METHOD PUBLIC CallAfterInit
VAR_INPUT
    AxisRef : REFERENCE TO AXIS_REF;
END_VAR
THIS^.AxisRef REF= AxisRef;
END_METHOD

{warning 'add property implementation'}
PROPERTY Done : BOOL
GET
Done := bDone;
END_GET
END_PROPERTY

{warning 'add property implementation'}
PROPERTY Error : BOOL
GET
Error := bError;
END_GET
END_PROPERTY

{warning 'add property implementation'}
PROPERTY ErrorID : UDINT
GET
ErrorID := nErrorID;
END_GET
END_PROPERTY

METHOD FB_Init : BOOL
VAR_INPUT
    bInitRetains : BOOL; // if TRUE, the retain variables are initialized (warm start / cold start)
    bInCopyCode : BOOL;  // if TRUE, the instance afterwards gets moved into the copy code (online change)
    AxisRef : REFERENCE TO AXIS_REF;
END_VAR
THIS^.AxisRef REF= AxisRef;
END_METHOD

PROPERTY Message : T_MAXSTRING
GET
Message :=sMessage;
END_GET
END_PROPERTY

METHOD Reset
VAR_INPUT
    Execute	: BOOL;
END_VAR
THIS^.bExecute := Execute;
END_METHOD

END_FUNCTION_BLOCK

// ---- POUs/FBs/NC/FB_HaltNC.TcPOU
FUNCTION_BLOCK FB_HaltNC IMPLEMENTS I_Halt
VAR_INPUT
    {attribute 'no_copy'}
    AxisRef : REFERENCE TO AXIS_REF;
    fbMcHalt 		: MC_Halt;
    bCommandHalt :BOOL;
    fDeceleration : LREAL;
    fJerk :LREAL;
    eBufferMode : MC_BufferMode := MC_BufferMode.MC_Aborting;
    bError : BOOL;
    bBusy : BOOL;
    bDone : BOOL;
    nErrorID : UDINT;
    sMessage : T_MAXSTRING;
    rtDone : R_TRIG;
    bAborted : BOOL;
END_VAR
VAR_OUTPUT
END_VAR
VAR
END_VAR

IF NOT __ISVALIDREF(THIS^.AxisRef) THEN
    RETURN;
END_IF

THIS^.AxisRef.ReadStatus();

THIS^.fbMcHalt(
    Axis := THIS^.AxisRef,
    Execute := THIS^.bCommandHalt,
    Deceleration := THIS^.fDeceleration,
    Jerk := THIS^.fJerk,
    BufferMode := THIS^.eBufferMode,
    Done =>THIS^.bDone,
    Busy => THIS^.bBusy,
    CommandAborted =>THIS^.bAborted,
    Error => THIS^.bError,
    ErrorID => THIS^.nErrorID
);

rtDone(CLK:=bDone);
IF  rtDone.Q THEN
    THIS^.bCommandHalt := FALSE;
END_IF

{warning 'Add property implementation'}
PROPERTY Aborted : BOOL
GET
Aborted := THIS^.bAborted;
END_GET
END_PROPERTY

{warning 'Add property implementation'}
PROPERTY Active : BOOL
GET
Active := THIS^.fbMcHalt.Active;
END_GET
END_PROPERTY

{warning 'add property implementation'}
PROPERTY Busy : BOOL
GET
Busy := bBusy;
END_GET
END_PROPERTY

METHOD PUBLIC CallAfterInit
VAR_INPUT
    AxisRef : REFERENCE TO AXIS_REF;
END_VAR
THIS^.AxisRef REF= AxisRef;
END_METHOD

PROPERTY CommandHalt : BOOL
SET
bCommandHalt := CommandHalt;
END_SET
END_PROPERTY

PROPERTY Done : BOOL
GET
Done := bDone;
END_GET
END_PROPERTY

{warning 'add property implementation'}
PROPERTY Error : BOOL
GET
Error := bError;
END_GET
END_PROPERTY

{warning 'add property implementation'}
PROPERTY ErrorID : UDINT
GET
ErrorID := nErrorID;
END_GET
END_PROPERTY

//FB_Init is always available implicitly and it is used primarily for initialization.
//The return value is not evaluated. For a specific influence, you can also declare the
//methods explicitly and provide additional code there with the standard initialization
//code. You can evaluate the return value.
METHOD FB_Init: BOOL
VAR_INPUT
    bInitRetains: BOOL; // TRUE: the retain variables are initialized (reset warm / reset cold)
    bInCopyCode: BOOL;  // TRUE: the instance will be copied to the copy code afterward (online change)
    AxisRef : REFERENCE TO AXIS_REF;
END_VAR
THIS^.AxisRef REF= AxisRef;
END_METHOD

METHOD Halt
VAR_INPUT
    Execute	: BOOL;
    Deceleration	: LREAL := 0;
    Jerk	: LREAL := 0;
    BufferMode	: MC_BufferMode := .MC_BufferMode.MC_Aborting;
END_VAR
THIS^.bCommandHalt :=  Execute;
THIS^.fDeceleration := Deceleration;
THIS^.fJerk := Jerk;
THIS^.eBufferMode := BufferMode;
END_METHOD

PROPERTY Message : T_MAXSTRING
GET
Message  := sMessage;
END_GET
END_PROPERTY

END_FUNCTION_BLOCK

// ---- Test/NC/FB_MotionAxisNC_Test.TcPOU
FUNCTION_BLOCK FB_MotionAxisNC_Test EXTENDS FB_TestSuite
VAR
	fbAxisRef : AXIS_REF;
	fbMotionLogger : FB_MotionLogger;
    fbHome : FB_HomeNC_TestDouble;
    fbHalt : FB_HaltNC_TestDouble;
    fbPower : FB_PowerNC_TestDouble;
    fbReset : FB_ResetNC_TestDouble;
    fbMoveAbsolute : FB_MoveAbsoluteNC_TestDouble;
    fbReadParameter : FB_ReadParameterNC_TestDouble;
    fbWriteParameter  : FB_WriteParameterNC_TestDouble;
    fbParamSaveRestore: FB_ParamSaveRestoreNC_TestDouble;
    fbEncoderScaling : FB_EncoderScalingNC_TestDouble;
    fbAxisStatus : FB_AxisStatusNC_TestDouble;
    fbBacklashCompensation : FB_BacklashCompensationNC_TestDouble;
END_VAR

GivenAllMCBlockErrorConditionThenPowerErrorHasHigherPriority();

METHOD PRIVATE GivenAllMCBlockErrorConditionThenPowerErrorHasHigherPriority
VAR_INST
    // subject under test
    // subject under test
    fbMotionAxis : FB_MotionAxisNC(  	
		AxisRef :=fbAxisRef,
		iMotionLogger := fbMotionLogger,
		iHome := fbHome,
        iHalt := fbHalt,
        iPower := fbPower,
        iReset := fbReset,
        iMoveAbsolute := fbMoveAbsolute,
        iReadParameter := fbReadParameter,
        iWriteParameter  := fbWriteParameter,
        iParamsSaveRestore:= fbParamSaveRestore,
        iEncoderScaling := fbEncoderScaling,
        iBacklashCompensation := fbBacklashCompensation
	);
bExpectedAxisError :BOOL := TRUE;
nExpectedErrorId: UDINT;
END_VAR
TEST(__POUNAME());
// ----- Power: Highest priority -----
fbHome.Error := TRUE;
fbHalt.Error := TRUE;
fbPower.Error := TRUE;
fbReset.Error := TRUE;
fbMoveAbsolute.Error := TRUE;
fbReadParameter.Error := TRUE;
fbWriteParameter.Error := TRUE;
fbParamSaveRestore.Error := TRUE;
fbBacklashCompensation.Error := TRUE;

fbMotionAxis();

AssertTrue(
    Condition := fbMotionAxis.Status.bError,
    Message   := 'Prioritized and generalized Error must be set #1'
);
AssertEquals_UDINT(
    Expected := 18000,
    Actual   := fbMotionAxis.Status.nErrorID,
    Message  := 'Prioritized error Id must be 18000 #2'
);

// ----- Halt: Second -----
fbPower.Error := FALSE;
fbHalt.Error := TRUE;
fbHome.Error := TRUE;
fbReset.Error := TRUE;
fbMoveAbsolute.Error := TRUE;
fbReadParameter.Error := TRUE;
fbWriteParameter.Error := TRUE;
fbParamSaveRestore.Error := TRUE;
fbBacklashCompensation.Error := TRUE;

fbMotionAxis();

AssertTrue(
    Condition := fbMotionAxis.Status.bError,
    Message   := 'Prioritized and generalized Error must be set #3'
);
AssertEquals_UDINT(
    Expected := 19000,
    Actual   := fbMotionAxis.Status.nErrorID,
    Message  := 'Prioritized error Id must be 19000 #4'
);

// ----- Reset: Third -----
fbPower.Error := FALSE;
fbHalt.Error := FALSE;
fbReset.Error := TRUE;
fbHome.Error := TRUE;
fbMoveAbsolute.Error := TRUE;
fbReadParameter.Error := TRUE;
fbWriteParameter.Error := TRUE;
fbParamSaveRestore.Error := TRUE;
fbBacklashCompensation.Error := TRUE;

fbMotionAxis();

AssertTrue(
    Condition := fbMotionAxis.Status.bError,
    Message   := 'Prioritized and generalized Error must be set #5'
);
AssertEquals_UDINT(
    Expected := 20000,
    Actual   := fbMotionAxis.Status.nErrorID,
    Message  := 'Prioritized error Id must be 20000 #6'
);

// ----- BacklashCompensation: Fourth -----
fbPower.Error := FALSE;
fbHalt.Error := FALSE;
fbReset.Error := FALSE;
fbBacklashCompensation.Error := TRUE;
fbHome.Error := TRUE;
fbMoveAbsolute.Error := TRUE;
fbReadParameter.Error := TRUE;
fbWriteParameter.Error := TRUE;
fbParamSaveRestore.Error := TRUE;

fbMotionAxis();

AssertTrue(
    Condition := fbMotionAxis.Status.bError,
    Message   := 'Prioritized and generalized Error must be set #7'
);
AssertEquals_UDINT(
    Expected := 21000,
    Actual   := fbMotionAxis.Status.nErrorID,
    Message  := 'Prioritized error Id must be 21000 #8'
);

// ----- MoveAbsolute: Fifth -----
fbBacklashCompensation.Error := FALSE;
fbMoveAbsolute.Error := TRUE;
fbPower.Error := FALSE;
fbHalt.Error := FALSE;
fbReset.Error := FALSE;
fbHome.Error := TRUE;
fbReadParameter.Error := TRUE;
fbWriteParameter.Error := TRUE;
fbParamSaveRestore.Error := TRUE;

fbMotionAxis();

AssertTrue(
    Condition := fbMotionAxis.Status.bError,
    Message   := 'Prioritized and generalized Error must be set #9'
);
AssertEquals_UDINT(
    Expected := 22000,
    Actual   := fbMotionAxis.Status.nErrorID,
    Message  := 'Prioritized error Id must be 22000 #10'
);

// ----- Home: Sixth -----
fbMoveAbsolute.Error := FALSE;
fbHome.Error := TRUE;
fbPower.Error := FALSE;
fbHalt.Error := FALSE;
fbReset.Error := FALSE;
fbBacklashCompensation.Error := FALSE;
fbReadParameter.Error := TRUE;
fbWriteParameter.Error := TRUE;
fbParamSaveRestore.Error := TRUE;

fbMotionAxis();

AssertTrue(
    Condition := fbMotionAxis.Status.bError,
    Message   := 'Prioritized and generalized Error must be set #11'
);
AssertEquals_UDINT(
    Expected := 23000,
    Actual   := fbMotionAxis.Status.nErrorID,
    Message  := 'Prioritized error Id must be 23000 #12'
);

// ----- ReadParameter: Eighth -----
fbHome.Error := FALSE;
fbReadParameter.Error := TRUE;
fbWriteParameter.Error := TRUE;
fbPower.Error := FALSE;
fbHalt.Error := FALSE;
fbReset.Error := FALSE;
fbBacklashCompensation.Error := FALSE;
fbMoveAbsolute.Error := FALSE;
fbParamSaveRestore.Error := TRUE;

fbMotionAxis();

AssertTrue(
    Condition := fbMotionAxis.Status.bError,
    Message   := 'Prioritized and generalized Error must be set #13'
);
AssertEquals_UDINT(
    Expected := 25000,
    Actual   := fbMotionAxis.Status.nErrorID,
    Message  := 'Prioritized error Id must be 25000 #14'
);

// ----- WriteParameter: Ninth -----
fbReadParameter.Error := FALSE;
fbWriteParameter.Error := TRUE;
fbPower.Error := FALSE;
fbHalt.Error := FALSE;
fbReset.Error := FALSE;
fbBacklashCompensation.Error := FALSE;
fbMoveAbsolute.Error := FALSE;
fbHome.Error := FALSE;
fbParamSaveRestore.Error := TRUE;

fbMotionAxis();

AssertTrue(
    Condition := fbMotionAxis.Status.bError,
    Message   := 'Prioritized and generalized Error must be set #15'
);
AssertEquals_UDINT(
    Expected := 26000,
    Actual   := fbMotionAxis.Status.nErrorID,
    Message  := 'Prioritized error Id must be 26000 #16'
);

// ----- ParamSaveRestore: Tenth -----
fbWriteParameter.Error := FALSE;
fbParamSaveRestore.Error := TRUE;
fbPower.Error := FALSE;
fbHalt.Error := FALSE;
fbReset.Error := FALSE;
fbBacklashCompensation.Error := FALSE;
fbMoveAbsolute.Error := FALSE;
fbHome.Error := FALSE;
fbReadParameter.Error := FALSE;

fbMotionAxis();

AssertTrue(
    Condition := fbMotionAxis.Status.bError,
    Message   := 'Prioritized and generalized Error must be set #17'
);
AssertEquals_UDINT(
    Expected := 27000,
    Actual   := fbMotionAxis.Status.nErrorID,
    Message  := 'Prioritized error Id must be 27000 #18'
);

TEST_FINISHED();
END_METHOD

END_FUNCTION_BLOCK

// ---- Test/TestDouble/FB_HomeNC_TestDouble.TcPOU
FUNCTION_BLOCK FB_HomeNC_TestDouble IMPLEMENTS I_Home
VAR
    bError : BOOL;
    nErrorID : UDINT := 23000;
END_VAR

PROPERTY Aborted : BOOL
GET
END_GET
END_PROPERTY

{warning 'Add method implementation '}
METHOD AbortRecovery
END_METHOD

PROPERTY Active : BOOL
GET
END_GET
END_PROPERTY

PROPERTY Busy : BOOL
GET
END_GET
END_PROPERTY

{warning 'Add method implementation '}
METHOD ClearStatus
END_METHOD

PROPERTY Done : BOOL
GET
END_GET
END_PROPERTY

PROPERTY Error : BOOL
GET
Error := bError;
END_GET
SET
bError := Error;
END_SET
END_PROPERTY

PROPERTY ErrorID : UDINT
GET
ErrorId := nErrorID;
END_GET
SET
nErrorId := ErrorID;
END_SET
END_PROPERTY

METHOD Home : BOOL
VAR_INPUT
    Position        : LREAL         := DEFAULT_HOME_POSITION;
    BufferMode      : MC_BufferMode;
 	HomeMode: INT :=E_EpicsHomeCmd.NONE;
END_VAR
END_METHOD

{warning 'Add method implementation '}
METHOD HomeDone
END_METHOD

PROPERTY LimHomeDone : BOOL
GET
END_GET
END_PROPERTY

PROPERTY Message : T_MAXSTRING
GET
END_GET
END_PROPERTY

PROPERTY Mode : INT
GET
END_GET
SET
END_SET
END_PROPERTY

PROPERTY Offset : LREAL
SET
END_SET
END_PROPERTY

PROPERTY Position : LREAL
SET
END_SET
END_PROPERTY

END_FUNCTION_BLOCK

// ---- Test/TestDouble/FB_HaltNC_TestDouble.TcPOU
FUNCTION_BLOCK FB_HaltNC_TestDouble IMPLEMENTS  I_Halt
VAR
	bError : BOOL;
	nErrorID : UDINT := 19000;
END_VAR

{warning 'Add property implementation'}
PROPERTY Aborted : BOOL
GET
END_GET
END_PROPERTY

{warning 'Add property implementation'}
PROPERTY Active : BOOL
GET
Active := TRUE;
END_GET
END_PROPERTY

{warning 'Add property implementation'}
PROPERTY Busy : BOOL
GET
END_GET
END_PROPERTY

{warning 'Add property implementation'}
PROPERTY CommandHalt : BOOL
SET
END_SET
END_PROPERTY

{warning 'Add property implementation'}
PROPERTY Done : BOOL
GET
END_GET
END_PROPERTY

{warning 'Add property implementation'}
PROPERTY Error : BOOL
GET
Error := bError;
END_GET
SET
bError := Error;
END_SET
END_PROPERTY

{warning 'Add property implementation'}
PROPERTY ErrorID : UDINT
GET
ErrorId := nErrorID;
END_GET
SET
nErrorId := ErrorID;
END_SET
END_PROPERTY

{warning 'Add method implementation '}
METHOD Halt
VAR_INPUT
	Deceleration	: LREAL := 0;
	Jerk	: LREAL := 0;
	BufferMode	: MC_BufferMode := .MC_BufferMode.MC_Aborting;
END_VAR
END_METHOD

{warning 'Add method implementation '}
METHOD HaltDone
END_METHOD

{warning 'Add property implementation'}
PROPERTY Message : T_MAXSTRING
GET
END_GET
END_PROPERTY

END_FUNCTION_BLOCK

// ---- Test/TestDouble/FB_PowerNC_TestDouble.TcPOU
FUNCTION_BLOCK FB_PowerNC_TestDouble IMPLEMENTS  I_Power
VAR
    bError : BOOL;
    nErrorID : UDINT := 18000;
END_VAR

PROPERTY Aborted : BOOL
GET
END_GET
END_PROPERTY

PROPERTY Active : BOOL
GET
END_GET
END_PROPERTY

PROPERTY Busy : BOOL
GET
END_GET
END_PROPERTY

{warning 'Add property implementation'}
PROPERTY DirectionalPowerEnabled : BOOL
GET
END_GET
END_PROPERTY

METHOD DisablePower
END_METHOD

PROPERTY Done : BOOL
GET
END_GET
END_PROPERTY

PROPERTY Error : BOOL
GET
Error := bError;
END_GET
SET
bError := Error;
END_SET
END_PROPERTY

PROPERTY ErrorID : UDINT
GET
ErrorId := nErrorID;
END_GET
SET
nErrorId := ErrorID;
END_SET
END_PROPERTY

PROPERTY Message : T_MAXSTRING
GET
END_GET
END_PROPERTY

PROPERTY Override : LREAL
GET
END_GET
END_PROPERTY

METHOD Power
VAR_INPUT
    Enable	: BOOL;
    Enable_Positive	: BOOL;
    Enable_Negative	: BOOL;
    Override	: LREAL := 100;
    BufferMode	: MC_BufferMode := MC_BufferMode.MC_Aborting;
END_VAR
END_METHOD

PROPERTY PowerIsEnabled : BOOL
GET
PowerIsEnabled := TRUE;
END_GET
END_PROPERTY

END_FUNCTION_BLOCK

// ---- Test/TestDouble/FB_ResetNC_TestDouble.TcPOU
FUNCTION_BLOCK FB_ResetNC_TestDouble IMPLEMENTS  I_Reset
VAR
	bError : BOOL;
	nErrorID : UDINT := 20000;
END_VAR

{warning 'Add property implementation'}
PROPERTY Aborted : BOOL
GET
END_GET
END_PROPERTY

{warning 'Add property implementation'}
PROPERTY Active : BOOL
GET
Active := TRUE;
END_GET
END_PROPERTY

{warning 'Add property implementation'}
PROPERTY Busy : BOOL
GET
END_GET
END_PROPERTY

{warning 'Add property implementation'}
PROPERTY Done : BOOL
GET
END_GET
END_PROPERTY

{warning 'Add property implementation'}
PROPERTY Error : BOOL
GET
Error := bError;
END_GET
SET
bError := Error;
END_SET
END_PROPERTY

{warning 'Add property implementation'}
PROPERTY ErrorID : UDINT
GET
ErrorId := nErrorID;
END_GET
SET
nErrorId := ErrorID;
END_SET
END_PROPERTY

{warning 'Add property implementation'}
PROPERTY Message : T_MAXSTRING
GET
END_GET
END_PROPERTY

{warning 'Add method implementation '}
METHOD Reset
END_METHOD

{warning 'Add method implementation '}
METHOD ResetDone
END_METHOD

END_FUNCTION_BLOCK

// ---- Test/TestDouble/FB_MoveAbsoluteNC_TestDouble.TcPOU
FUNCTION_BLOCK FB_MoveAbsoluteNC_TestDouble IMPLEMENTS I_MoveABsolute
VAR
    bError : BOOL;
    nErrorID : UDINT := 22000;
END_VAR

PROPERTY Aborted : BOOL
GET
END_GET
END_PROPERTY

PROPERTY Active : BOOL
GET
END_GET
END_PROPERTY

PROPERTY Busy : BOOL
GET
END_GET
END_PROPERTY

PROPERTY CommandMoveAbsolute : BOOL
SET
END_SET
END_PROPERTY

PROPERTY Done : BOOL
GET
END_GET
END_PROPERTY

PROPERTY Error : BOOL
GET
Error := bError;
END_GET
SET
bError := Error;
END_SET
END_PROPERTY

PROPERTY ErrorID : UDINT
GET
ErrorId := nErrorID;
END_GET
SET
nErrorId := ErrorID;
END_SET
END_PROPERTY

PROPERTY Message : T_MAXSTRING
GET
END_GET
END_PROPERTY

METHOD MoveAbsolute
VAR_INPUT
    Position	: LREAL;
    Velocity	: LREAL;
    Acceleration	: LREAL := 0;
    Deceleration	: LREAL := 0;
    Jerk	: LREAL := 0;
    BufferMode	: MC_BufferMode := MC_BufferMode.MC_Aborting;
END_VAR
END_METHOD

{warning 'Add method implementation '}
METHOD MoveAbsoluteDone
END_METHOD

END_FUNCTION_BLOCK

// ---- Test/TestDouble/FB_WriteParameterNC_TestDouble.TcPOU
FUNCTION_BLOCK FB_WriteParameterNC_TestDouble IMPLEMENTS  I_WriteParameter
VAR
	bError : BOOL;
	nErrorID : UDINT := 26000;
END_VAR

{warning 'Add property implementation'}
PROPERTY Aborted : BOOL
GET
END_GET
END_PROPERTY

{warning 'Add property implementation'}
PROPERTY Active : BOOL
GET
END_GET
END_PROPERTY

{warning 'Add property implementation'}
PROPERTY Busy : BOOL
GET
END_GET
END_PROPERTY

{warning 'Add property implementation'}
PROPERTY Done : BOOL
GET
END_GET
END_PROPERTY

{warning 'Add property implementation'}
PROPERTY Error : BOOL
GET
Error := bError;
END_GET
SET
bError := Error;
END_SET
END_PROPERTY

{warning 'Add property implementation'}
PROPERTY ErrorID : UDINT
GET
ErrorId := nErrorID;
END_GET
SET
nErrorId := ErrorID;
END_SET
END_PROPERTY

{warning 'Add property implementation'}
PROPERTY Message : T_MAXSTRING
GET
END_GET
END_PROPERTY

{warning 'Add method implementation '}
METHOD WriteParameter
VAR_INPUT
	ParameterNumber	: MC_AxisParameter;
	ParameterValue	: LREAL;
END_VAR
END_METHOD

END_FUNCTION_BLOCK

// ---- Test/TestDouble/FB_AxisStatusNC_TestDouble.TcPOU
FUNCTION_BLOCK FB_AxisStatusNC_TestDouble IMPLEMENTS I_AxisStatus
VAR
	bError : BOOL;
	nErrorID : UDINT := 24000;
END_VAR

{warning 'Add property implementation'}
PROPERTY Aborted : BOOL
GET
END_GET
END_PROPERTY

{warning 'Add property implementation'}
PROPERTY Active : BOOL
GET
END_GET
END_PROPERTY

{warning 'Add method implementation '}
METHOD AxisEnabled : BOOL
END_METHOD

{warning 'Add property implementation'}
PROPERTY AxisID : UDINT
GET
END_GET
END_PROPERTY

{warning 'Add property implementation'}
PROPERTY AxisState : MC_AxisStates
GET
END_GET
END_PROPERTY

{warning 'Add property implementation'}
PROPERTY Busy : BOOL
GET
END_GET
END_PROPERTY

{warning 'Add property implementation'}
PROPERTY Done : BOOL
GET
END_GET
END_PROPERTY

{warning 'Add property implementation'}
PROPERTY Error : BOOL
GET
Error := bError;
END_GET
SET
bError := Error;
END_SET
END_PROPERTY

{warning 'Add property implementation'}
PROPERTY ErrorID : UDINT
GET
ErrorId := nErrorID;
END_GET
SET
nErrorId := ErrorID;
END_SET
END_PROPERTY

{warning 'Add property implementation'}
PROPERTY InTargetPosition : BOOL
GET
END_GET
END_PROPERTY

{warning 'Add property implementation'}
PROPERTY MeasuredAcceleration : LREAL
GET
END_GET
END_PROPERTY

{warning 'Add property implementation'}
PROPERTY MeasuredPosition : LREAL
GET
END_GET
END_PROPERTY

{warning 'Add property implementation'}
PROPERTY MeasuredPositionDiff : LREAL
GET
END_GET
END_PROPERTY

{warning 'Add property implementation'}
PROPERTY MeasuredVelocity : LREAL
GET
END_GET
END_PROPERTY

{warning 'Add property implementation'}
PROPERTY Message : T_MAXSTRING
GET
END_GET
END_PROPERTY

{warning 'Add property implementation'}
PROPERTY NegativeMotionIsEnabled : BOOL
GET
END_GET
END_PROPERTY

{warning 'Add property implementation'}
PROPERTY PositiveMotionIsEnabled : BOOL
GET
END_GET
END_PROPERTY

{warning 'Add property implementation'}
PROPERTY StandStill : BOOL
GET
END_GET
END_PROPERTY

{warning 'Add property implementation'}
PROPERTY Stopped : BOOL
GET
END_GET
END_PROPERTY

END_FUNCTION_BLOCK

// ---- Test/TestDouble/FB_BacklashCompensationNC_TestDouble.TcPOU
FUNCTION_BLOCK FB_BacklashCompensationNC_TestDouble IMPLEMENTS I_BacklashCompensation
VAR
    bError : BOOL;
    nErrorID : UDINT := 21000;
END_VAR

METHOD BacklashCompensation
VAR_INPUT
    Enable	: BOOL := FALSE;
    RampVelo	: LREAL;
END_VAR
END_METHOD

METHOD BacklashCompensationTest
VAR_INPUT
    UserEnable	: BOOL;
    Compensation	: LREAL;
END_VAR
END_METHOD

PROPERTY Busy : BOOL
GET
END_GET
END_PROPERTY

{warning 'Add method implementation '}
METHOD ClearStatus
END_METHOD

PROPERTY CurrentBacklash : LREAL
GET
END_GET
END_PROPERTY

PROPERTY Enable : BOOL
SET
END_SET
END_PROPERTY

{warning 'Add method implementation '}
METHOD EnableBacklashCompensation
VAR_INPUT
	UserEnable	: BOOL;
	Compensation	: LREAL;
END_VAR
END_METHOD

PROPERTY Error : BOOL
GET
Error := bError;
END_GET
SET
bError := Error;
END_SET
END_PROPERTY

PROPERTY ErrorID : UDINT
GET
ErrorId := nErrorID;
END_GET
SET
nErrorId := ErrorID;
END_SET
END_PROPERTY

PROPERTY Message : T_MAXSTRING
GET
END_GET
END_PROPERTY

PROPERTY Status : BOOL
GET
END_GET
END_PROPERTY

PROPERTY UserEnable : BOOL
SET
END_SET
END_PROPERTY

END_FUNCTION_BLOCK

// ---- POUs/FBs/NC/FB_MotionAxisNC.TcPOU
FUNCTION_BLOCK FB_MotionAxisNC IMPLEMENTS I_MotionAxis
VAR_INPUT
END_VAR
VAR_OUTPUT
END_VAR
VAR
    iHome : I_Home;
    iHalt : I_Halt;
    iPower : I_Power;
    iReset : I_Reset;
    iMoveAbsolute : I_MoveAbsolute;
    iReadParameter : I_ReadParameter;
    iWriteParameter  : I_WriteParameter;
    iParamSaveRestore: I_ParamSaveRestore;
    iEncoderScaling : I_EncoderScaling;
    iAxisStatus : I_AxisStatus;
    iBacklashCompensation : I_BacklashCompensation;

     bError: BOOL;
     nErrorID: UDINT;
     sMessage : T_MAXSTRING;
     rtAbortDone : R_TRIG;

END_VAR

// Forward the abort event to homing block ( this is to sync the home state machine)
// Clear local execs flags after a completed move or a completed interruption
rtAbortDone(CLK:=(THIS^.iHalt.Done OR THIS^.iReset.Done));
IF  rtAbortDone.Q THEN
    THIS^.iMoveAbsolute.CommandMoveAbsolute := FALSE;
    THIS^.iHome.CommandMoveHome := FALSE;
    // forward global reset done event;
    THIS^.iHome.GlobalReset := THIS^.iReset.Done;
END_IF

// handle combined Errors conditions
THIS^.ErrorHandling();

PROPERTY AbortDone : BOOL
GET
AbortDone := THIS^.iHalt.Done OR THIS^.iReset.Done;
END_GET
END_PROPERTY

PROPERTY Aborted : BOOL
GET
ABorted := THIS^.iMoveAbsolute.Aborted;
END_GET
END_PROPERTY

METHOD AxisEnabled : BOOL
VAR_INPUT
    HomeCmd : BOOL;
    NewMoveReq : BOOL;
END_VAR
AxisEnabled:=THIS^.iAxisStatus.AxisEnabled();
END_METHOD

PROPERTY AxisReadParamsInit : BOOL
GET
AxisReadParamsInit := THIS^.iReadParameter.AxisReadParamsInit;
END_GET
END_PROPERTY

PROPERTY AxisState : MC_AxisStates
GET
AxisState := THIS^.iAxisStatus.AxisState;
END_GET
END_PROPERTY

(*
    Handle positive/negative backlash compensation
    User needs to set the direction of backlash from the sign of the compensation value
    Backlash compensation is disabled during referencing (homing).
    When direction is positive/negative, further movement in the negative/positive direction not compensated
    further movement in the negative/positive direction will be compensated
*)
METHOD BacklashCompensation
VAR_INPUT
    Active     : BOOL;
    Compensation	: LREAL;
    RampVelocity	: LREAL;
    DisableMode	: E_DISABLEMODE := E_DISABLEMODE.DisableModeHold;
END_VAR
THIS^.iBacklashCompensation.BacklashCompensation(	Activate:=Active,
                                                    Compensation:=Compensation,
                                                    RampVelocity:=RampVelocity,
                                                    DisableMode:=DisableMode
                                                );
END_METHOD

(*synced Fbs need just to activate the compensation with a given ramp speed
  other parameters are provided via EPICS (declared in this FB) or via the more extended BackalshCompensation method (simulation) *)
METHOD BacklashCompensationActive
VAR_INPUT
    Active	: BOOL;
    RampVelocity	: LREAL;
END_VAR
THIS^.iBacklashCompensation.BacklashCompensationActive( Active:=Active,
                                                        RampVelocity:=RampVelocity );
END_METHOD

{warning 'Add property implementation'}
PROPERTY BacklashCompStatus : BOOL
GET
END_GET
END_PROPERTY

PROPERTY BacklashCompUserEn : BOOL
SET
THIS^.iBacklashCompensation.UserEnable:=BacklashCompUserEn;
END_SET
END_PROPERTY

PROPERTY Busy : BOOL
GET
Busy := THIS^.iHome.Busy OR THIS^.iMoveAbsolute.Busy;
END_GET
END_PROPERTY

METHOD PUBLIC CallAfterInit
VAR_INPUT
    iHome : I_Home;
    iHalt : I_Halt;
    iPower : I_Power;
    iReset : I_Reset;
    iMoveAbsolute : I_MoveAbsolute;
    iReadParameter : I_ReadParameter;
    iWriteParameter  : I_WriteParameter;
    iParamSaveRestore: I_ParamSaveRestore;
    iEncoderScaling : I_EncoderScaling;
    iAxisStatus : I_AxisStatus;
    iBacklashCompensation : I_BacklashCompensation;
END_VAR
THIS^.iHome := iHome;
THIS^.iHalt := iHalt;
THIS^.iPower := iPower;
THIS^.iReset := iReset;
THIS^.iMoveAbsolute := iMoveAbsolute;
THIS^.iReadParameter := iReadParameter ;
THIS^.iWriteParameter  := iWriteParameter;
THIS^.iParamSaveRestore:= iParamSaveRestore;
THIS^.iEncoderScaling := iEncoderScaling;
THIS^.iAxisStatus := iAxisStatus;
THIS^.iBacklashCompensation  := iBacklashCompensation ;
END_METHOD

PROPERTY Done : BOOL
GET
Done := THIS^.iHome.Done OR THIS^.iMoveAbsolute.Done;
END_GET
END_PROPERTY

PROPERTY Error : BOOL
GET
Error := bError;
END_GET
END_PROPERTY

METHOD ErrorHandling
(*
    Error from functions and Nc
    The error will send to EPICS interface based on predifined
    priority: axis, power, backlash, absoluteMove, etc...
*)
IF THIS^.iAxisStatus.Error  THEN
    bError:=THIS^.iAxisStatus.Error;
    nErrorId:=THIS^.iAxisStatus.ErrorID;
    sMessage := THIS^.iAxisStatus.Message;
ELSIF THIS^.iPower.Error AND THIS^.iPower.IsEnabled THEN
    bError:=THIS^.iPower.Error;
    nErrorId:=THIS^.iPower.ErrorID;
    sMessage := THIS^.iPower.Message;
ELSIF THIS^.iBacklashCompensation.Error THEN
    bError:=THIS^.iBacklashCompensation.Error;
    nErrorId:=THIS^.iBacklashCompensation.ErrorID;
    sMessage := THIS^.iBacklashCompensation.Message;
ELSIF THIS^.iMoveAbsolute.Error THEN
    bError:=THIS^.iMoveAbsolute.Error;
    nErrorId:=THIS^.iMoveAbsolute.ErrorID;
    sMessage := THIS^.iMoveAbsolute.Message;
ELSIF THIS^.iHome.Error (*Homing error*) THEN
    bError:=THIS^.iHome.Error;
    nErrorId:=THIS^.iHome.ErrorID;
    sMessage := THIS^.iHome.Message;
ELSIF THIS^.iHalt.Error AND THIS^.iHalt.Active THEN
    bError:=THIS^.iHalt.Error;
    nErrorId:=THIS^.iHalt.ErrorID;
    sMessage := THIS^.iHalt.Message;
ELSIF THIS^.iReset.Error  THEN
    bError:=THIS^.iReset.Error;
    nErrorId:=THIS^.iReset.ErrorID;
    sMessage := THIS^.iReset.Message;
ELSIF THIS^.iReadParameter.Error THEN
    bError := THIS^.iReadParameter.Error;
    nErrorId := THIS^.iReadParameter.ErrorID;
    sMessage := THIS^.iReadParameter.Message;
ELSIF THIS^.iWriteParameter.Error THEN
    bError := THIS^.iWriteParameter.Error;
    nErrorId := THIS^.iWriteParameter.ErrorID;
    sMessage := THIS^.iWriteParameter.Message;
ELSIF THIS^.iParamSaveRestore.Error THEN
    bError := THIS^.iParamSaveRestore.Error;
    nErrorId := THIS^.iParamSaveRestore.ErrorID;
    sMessage := THIS^.iParamSaveRestore.Message;
ELSE
    bError:=FALSE;
    nErrorId:=0;
    sMessage := '';
END_IF;
END_METHOD

PROPERTY ErrorID : UDINT
GET
ErrorID := THIS^.nErrorID;
END_GET
END_PROPERTY

//FB_Init is always available implicitly and it is used primarily for initialization.
//The return value is not evaluated. For a specific influence, you can also declare the
//methods explicitly and provide additional code there with the standard initialization
//code. You can evaluate the return value.
METHOD FB_Init: BOOL
VAR_INPUT
    bInitRetains: BOOL; // TRUE: the retain variables are initialized (reset warm / reset cold)
    bInCopyCode: BOOL;  // TRUE: the instance will be copied to the copy code afterward (online change)

    iHome : I_Home;
    iHalt : I_Halt;
    iPower : I_Power;
    iReset : I_Reset;
    iMoveAbsolute : I_MoveAbsolute;
    iReadParameter : I_ReadParameter;
    iWriteParameter  : I_WriteParameter;
    iParamSaveRestore: I_ParamSaveRestore;
    iEncoderScaling : I_EncoderScaling;
    iAxisStatus : I_AxisStatus;
    iBacklashCompensation : I_BacklashCompensation;
END_VAR
THIS^.iHome := iHome;
THIS^.iHalt := iHalt;
THIS^.iPower := iPower;
THIS^.iReset := iReset;
THIS^.iMoveAbsolute := iMoveAbsolute;
THIS^.iReadParameter := iReadParameter ;
THIS^.iWriteParameter  := iWriteParameter;
THIS^.iParamSaveRestore:= iParamSaveRestore;
THIS^.iEncoderScaling := iEncoderScaling;
THIS^.iAxisStatus := iAxisStatus;
THIS^.iBacklashCompensation  := iBacklashCompensation ;
END_METHOD

METHOD Halt
VAR_INPUT
    Execute	: BOOL;
    Deceleration	: LREAL := 0;
    Jerk	: LREAL := 0;
    BufferMode	: MC_BufferMode := MC_BufferMode.MC_Aborting;
END_VAR
THIS^.iHalt.Halt( Execute:=Execute,
                     Deceleration:=Deceleration,
                    Jerk:=Jerk ,
                    BufferMode:=BufferMode );
END_METHOD

{warning 'Add property implementation'}
PROPERTY HaltActive : BOOL
GET
END_GET
END_PROPERTY

{warning 'Add property implementation'}
PROPERTY HaltBusy : BOOL
GET
END_GET
END_PROPERTY

PROPERTY HaltDone : BOOL
GET
HaltDone := THIS^.iHalt.Done;
END_GET
END_PROPERTY

METHOD Home
VAR_INPUT
    Execute	: BOOL;
    HomeSpeedFast	: LREAL;
    HomeSpeedSlow	: LREAL;
END_VAR
//
THIS^.iHome.Home( Execute:=Execute,
                  HomeSpeedFast:=HomeSpeedFast,
                  HomeSpeedSlow:=HomeSpeedSlow );
END_METHOD

PROPERTY HomeBusy : BOOL
GET
HomeBusy := THIS^.iHome.Busy;
END_GET
END_PROPERTY

PROPERTY HomeDone : BOOL
GET
HomeDone := THIS^.iHome.Done;
END_GET
END_PROPERTY

{warning 'Add property implementation'}
PROPERTY HomeMode : E_EpicsHomeCmd
GET
HomeMode := THIS^.iHome.Mode;
END_GET
END_PROPERTY

PROPERTY InTargetPosition : BOOL
GET
InTargetPosition := THIS^.iAxisStatus.InTargetPosition;
END_GET
END_PROPERTY

PROPERTY MeasuredAcceleration : LREAL
GET
MeasuredAcceleration := THIS^.iAxisStatus.MeasuredAcceleration;
END_GET
END_PROPERTY

PROPERTY MeasuredCompensation : LREAL
GET
MeasuredCompensation := THIS^.iBacklashCompensation.ActCompensation;
END_GET
END_PROPERTY

PROPERTY MeasuredPosition : LREAL
GET
MeasuredPosition := THIS^.iAxisStatus.MeasuredPosition;
END_GET
END_PROPERTY

PROPERTY MeasuredPositionDiff : LREAL
GET
MeasuredPositionDiff := THIS^.iAxisStatus.MeasuredPositionDiff;
END_GET
END_PROPERTY

PROPERTY MeasuredVelocity : LREAL
GET
MeasuredVelocity := THIS^.iAxisStatus.MeasuredVelocity;
END_GET
END_PROPERTY

PROPERTY Message : T_MaxString
GET
Message :=sMessage;
END_GET
END_PROPERTY

METHOD MoveAbsolute
VAR_INPUT
    Execute     : BOOL;
    Position	: LREAL;
    Velocity	: LREAL;
    Acceleration	: LREAL := 0.0;
    Deceleration	: LREAL := 0.0;
    Jerk	: LREAL := 0.0;
    BufferMode	: MC_BufferMode := MC_BufferMode.MC_Aborting;
END_VAR
THIS^.iMoveAbsolute.MoveAbsolute( 	Execute:=Execute,
                                    Position:=Position,
                                       Velocity := Velocity,
                                    Acceleration := Acceleration,
                                    Deceleration := Deceleration,
                                    Jerk := Jerk,
                                    BufferMode := BufferMode);
END_METHOD

{warning 'Add property implementation'}
PROPERTY MoveAbsoluteAborted : BOOL
GET
MoveAbsoluteAborted := THIS^.iMoveAbsolute.Aborted;
END_GET
END_PROPERTY

{warning 'Add property implementation'}
PROPERTY MoveAbsoluteActive : BOOL
GET
END_GET
END_PROPERTY

PROPERTY MoveAbsoluteBusy : BOOL
GET
MoveAbsoluteBusy := THIS^.iMoveAbsolute.Busy;
END_GET
END_PROPERTY

{warning 'Add property implementation'}
PROPERTY MoveAbsoluteDone : BOOL
GET
MoveAbsoluteDone := THIS^.iMoveAbsolute.Done;
END_GET
END_PROPERTY

PROPERTY NegativeMotionIsEnabled : BOOL
GET
 NegativeMotionIsEnabled := THIS^.iAxisStatus.NegativeMotionIsEnabled;
END_GET
END_PROPERTY

PROPERTY PositiveMotionIsEnabled : BOOL
GET
PositiveMotionIsEnabled := THIS^.iAxisStatus.PositiveMotionIsEnabled;
END_GET
END_PROPERTY

METHOD Power
VAR_INPUT
    Enable	: BOOL;
    Enable_Positive	: BOOL;
    Enable_Negative	: BOOL;
    Override	: LREAL := 100.0;
    BufferMode	: MC_BufferMode := MC_BufferMode.MC_Aborting;
END_VAR
THIS^.iPower.Power(	Enable:=Enable,
                    Enable_Positive:= Enable_Positive,
                    Enable_Negative:=Enable_Negative,
                    Override:=Override,
                    BufferMode:=BufferMode
                );
END_METHOD

{warning 'Add property implementation'}
PROPERTY PowerActive : BOOL
GET
END_GET
END_PROPERTY

(*This is overriden by this object internal acess to the interlock instance
  this is intended to pass power enable flags via the fbMotionDrive
*)
METHOD PowerEnables
VAR_INPUT
    Enable	: BOOL;
    Enable_Positive	: BOOL;
    Enable_Negative	: BOOL;
END_VAR
THIS^.iPower.Power(	Enable:=Enable,
                    Enable_Positive:= Enable_Positive,
                    Enable_Negative:=Enable_Negative,
                    Override:=100.0,
                    BufferMode:=MC_BufferMode.MC_Aborting
                );
END_METHOD

PROPERTY PowerIsEnabled : BOOL
GET
END_GET
END_PROPERTY

{warning 'Add property implementation'}
PROPERTY PowerOverride : LREAL
GET
PowerOverride := THIS^.iPower.Override;
END_GET
END_PROPERTY

METHOD ReadAxisParams
VAR_INPUT
    Enable	: BOOL;
    RefreshDelay	: TIME;
END_VAR
THIS^.iReadParameter.ReadParameters(Enable:=Enable, RefreshDelay:=RefreshDelay);
END_METHOD

METHOD Reset
VAR_INPUT
    Execute	: BOOL;
END_VAR
THIS^.iReset.Reset(Execute:=Execute);
END_METHOD

PROPERTY ResetBusy : BOOL
GET
ResetBusy := THIS^.iReset.Busy;
END_GET
END_PROPERTY

PROPERTY ResetDone : BOOL
GET
ResetDone := THIS^.iReset.Done;
END_GET
END_PROPERTY

PROPERTY RestoreDone : BOOL
GET
RestoreDone := THIS^.iParamSaveRestore.RestoreDone;
END_GET
END_PROPERTY

METHOD SaveAxisParams
VAR_INPUT
    Enable	: BOOL;
END_VAR
THIS^.iParamSaveRestore.SaveAxisParams(Enable:=Enable);
END_METHOD

PROPERTY SavedPosition : LREAL
GET
SavedPosition := THIS^.iParamSaveRestore.SavedPosition;
END_GET
END_PROPERTY

PROPERTY ScaledEncoderCount : UDINT
GET
ScaledEncoderCount := THIS^.iEncoderScaling.EncoderCount;
END_GET
END_PROPERTY

{warning 'Add property implementation'}
PROPERTY StandStill : BOOL
GET
StandStill := THIS^.iAxisStatus.StandStill;
END_GET
END_PROPERTY

(*
    Check all post condition before updating bCommandedMoveAbsolute
    The implmentatation will depend on the axis type
    DS402 NC/Direct axis : Implementation need to check that the drive is in the correct mode before initaiting the move then set bCommandedMoveAbsolute
    MP NC axis : will immediately write to bCommandedMoveAbsolute
*)
METHOD StartMove
VAR_INPUT
    MoveMode	: E_EpicsMotorCmd;
    CmdExecute	: BOOL;
END_VAR
CASE MoveMode  OF
    E_EpicsMotorCmd.MOVE_ABSOLUTE:
       THIS^.iMoveAbsolute.CommandMoveAbsolute := CmdExecute;
    E_EpicsMotorCmd.HOME:
        THIS^.iHome.Home( Execute:=CmdExecute,
                            HomeSpeedFast:=THIS^.iReadParameter.RefVeloSearch,
                            HomeSpeedSlow:=THIS^.iReadParameter.RefVeloSync );
END_CASE
// for typical NC axis no further tests needed
//StartMove := CmdExecute;
END_METHOD

PROPERTY Stopped : BOOL
GET
Stopped := THIS^.iAxisStatus.Stopped;
END_GET
END_PROPERTY

END_FUNCTION_BLOCK

// ---- Test/Containers/FB_MotionStageNC_Test.TcPOU
FUNCTION_BLOCK INTERNAL FB_MotionStageNC_Test EXTENDS FB_TestSuite
VAR
    fbMotionLogger : ARRAY[1..17] OF FB_MotionLogger;
    fbPersistentDataStorage :  ARRAY[1..17] OF FB_PersistentDataStorage;
 	fbAxisRef :   ARRAY[1..17] OF AXIS_REF;
END_VAR

GivenMoveCmdAndMoveOkIfResetThenAbortMove_Test1();
GivenMoveCmdAndMoveOkIfHaltThenAbortMove_Test2();
GivenMoveCmdAndMoveOkMoveToTarget1ThenTarget2_Test3();
GivenMoveCmdAndValidInterlocksThenMoveToTarget_Test4();
GivenMoveCmdValidInterlockAndWrongMotionParamsThenGotoErrorStateIfResetThenGotoInitState_Test5();
GivenMoveCmdAndMoveOkAndPositiveBacklashEnabledThenMoveToTargetWithCompensation_Test6();
GivenMoveCmdAndMoveOkAndNegativeBacklashEnabledThenMoveToTargetWithCompensation_Test7();
GivenHomeCmdAndAbsoluteSetAndMoveOkThenMoveToUserDefinedHomePosition_Test8();
GivenHomeCmdNoneAndMoveOkThenSetHomeFlag_Test9();
GivenHomeCmdLowLimitModeBackwardSwPulseMoveOkThenMoveToUserDefinedHomePosition_Test10();
GivenHomeCmdHighLimitModeForwardSwPulseMoveOkThenMoveToUserDefinedHomePosition_Test11();
GivenHomeCmdHomeViaLowModeHomeSwPulseMoveOkThenMoveToUserDefinedHomePosition_Test12();
GivenHomeCmdHomeViaHighModeHomeSwPulseMoveOkThenMoveToUserDefinedHomePosition_Test13();
GivenHomeCmdHomeViaHighModeForwardSwPulseBeforeHomeSwPulseThenMoveToUserDefinePosition_Test14();
GivenHomeCmdHomeViaLowModeBackwardSwPulseBeforeHomeSwPulseThenMoveToUserDefinePosition_Test15();
GivenHomeCmdLowLimitModeAndResetThenAbortHoming_Test16();
OverallStageFeaturesAndOperationalTests_Test17();

METHOD PRIVATE GivenHomeCmdAndAbsoluteSetAndMoveOkThenMoveToUserDefinedHomePosition_Test8
VAR_INST
   fbMotionStage : FB_MotionStageNC(	sName := 'Test8',
                                        AxisRef := fbAxisRef[8],
                                        iMotionLogger := fbMotionLogger[8],
                                        iPersistentDataStorage := fbPersistentDataStorage[8]
                                    ) :=(SaveAxisParams := FALSE);
									
    fbTestTimer: TON := (IN:=TRUE, PT:=T#10S);
    nTestStep : INT;
END_VAR
TEST(__POUNAME());


CASE nTestStep OF
    0:
			// Enable safety interlocks and hardware limits
        fbMotionStage.EnableLimits(
			BackwardEnable:=TRUE, 
			ForwardEnable:=TRUE,
			HomeEnable:=FALSE
		);
        fbMotionStage.EnableInterlocks();
		nTestStep := 1;
	1:
		fbMotionStage.Home(HomePosition:=20.0, HomeMode:=E_EPicsHomeCmd.ABSOLUTE_SET);
		nTestStep := 2;
	2:
		IF fbMotionStage.stMotionStatus.bDone THEN
			AssertTrue(Condition :=(fbMotionStage.stMotionCommand.fHomePosition - fbAxisRef[8].NcToPlc.ActPos) = 0, Message := 'Hone position not set #1');
			nTestStep := 3;
		END_IF	
END_CASE

fbTestTimer();
fbMotionStage();

IF nTestStep = 3 THEN

TEST_FINISHED();
ELSIF fbTestTimer.Q THEN
    AssertTrue(
        Condition := FALSE,
        Message := CONCAT('Timed out at step: ', TO_STRING(nTestStep))
    );
    TEST_FINISHED();
END_IF
END_METHOD

METHOD PRIVATE GivenHomeCmdHighLimitModeForwardSwPulseMoveOkThenMoveToUserDefinedHomePosition_Test11
VAR_INST
   fbMotionStage : FB_MotionStageNC(	sName := 'Test11',
                                        AxisRef := fbAxisRef[11],
                                        iMotionLogger := fbMotionLogger[11],
                                        iPersistentDataStorage := fbPersistentDataStorage[11]
                                    ) :=(SaveAxisParams := FALSE);
									
    fbTestTimer: TON := (IN:=TRUE, PT:=T#10S);
    fbCamSwitchPulserSearch: TON := (IN:=TRUE, PT:=T#500MS);
    fbCamSwitchPulserSync: TON := (PT:=T#1000MS);
    nTestStep : INT;
END_VAR
TEST(__POUNAME());

CASE nTestStep OF
    0: // Enable all interlocks/limits to be ready for homing
        fbMotionStage.EnableLimits(
			BackwardEnable:=TRUE, 
			ForwardEnable:=TRUE,
			HomeEnable:=FALSE
		);
        fbMotionStage.EnableInterlocks();
        nTestStep := 1;

    1: // Issue home command (to low limit)
        fbMotionStage.Home(HomePosition := 20.0, HomeMode := E_EpicsHomeCmd.HIGH_LIMIT);
        nTestStep := 2;

    2: // Simulate limit switch drop/restore with cam switch events
        IF fbCamSwitchPulserSearch.Q THEN
			// simulate limit release
			fbMotionStage.EnableLimits(
				BackwardEnable:=TRUE, 
				ForwardEnable:=FALSE,
				HomeEnable:=FALSE
			);
            fbCamSwitchPulserSearch.IN := FALSE;
            fbCamSwitchPulserSync.IN := TRUE;
            nTestStep := 3;
        END_IF

    3: // Restore limit after cam event
        IF fbCamSwitchPulserSync.Q THEN
			fbMotionStage.EnableLimits(
				BackwardEnable:=TRUE, 
				ForwardEnable:=TRUE,
				HomeEnable:=FALSE
			);
            nTestStep := 4;
        END_IF

    4: // Wait for home sequence completion
        IF fbMotionStage.stMotionStatus.bDone THEN
            nTestStep := 5;
        END_IF
END_CASE

fbCamSwitchPulserSearch();
fbCamSwitchPulserSync();
fbTestTimer();
fbMotionStage();

IF nTestStep = 5 THEN
    AssertTrue(
        Condition := fbAxisRef[11].Status.Homed,
        Message := 'Axis not calibrated #1'
    );
    AssertEquals_LREAL(
        Delta := 0.001,
        Expected := fbMotionStage.stMotionCommand.fHomePosition,
        Actual := fbAxisRef[11].NcToPlc.ActPos,
        Message := 'Position is not the expected #2'
    );
    TEST_FINISHED();
ELSIF fbTestTimer.Q THEN
    AssertTrue(
        Condition := FALSE,
        Message := CONCAT('Timed out at step: ', TO_STRING(nTestStep))
    );
    TEST_FINISHED();
END_IF
END_METHOD

METHOD PRIVATE GivenHomeCmdHomeViaHighModeForwardSwPulseBeforeHomeSwPulseThenMoveToUserDefinePosition_Test14
VAR_INST
   fbMotionStage : FB_MotionStageNC(	sName := 'Test14',
                                        AxisRef := fbAxisRef[14],
                                        iMotionLogger := fbMotionLogger[14],
                                        iPersistentDataStorage := fbPersistentDataStorage[14]
                                    ) :=(SaveAxisParams := FALSE);
									
    fbTestTimer: TON := (IN:=TRUE, PT:=T#10S);
    fbCamSwitchPulserSearch: TON := (IN:=TRUE, PT:=T#500MS);
    fbCamSwitchPulserSync: TON := (PT:=T#1000MS);
    nTestStep : INT;
END_VAR
TEST(__POUNAME());

CASE nTestStep OF
    0: // Enable all interlocks/limits for initial homing (home switch not active yet!)
        fbMotionStage.EnableLimits(
            BackwardEnable := TRUE, 
            ForwardEnable  := TRUE,
            HomeEnable     := FALSE
        );
        fbMotionStage.EnableInterlocks();
        nTestStep := 1;

    1: // Issue homing command (via high limit, should travel to positive end first)
        fbMotionStage.Home(
            HomePosition := 5.0,
            HomeMode := E_EpicsHomeCmd.HOME_VIA_HIGH
        );
        nTestStep := 2;

    2: // Simulate forward limit drop
        IF fbCamSwitchPulserSearch.Q THEN
            fbMotionStage.EnableLimits(
                BackwardEnable := TRUE, 
                ForwardEnable  := FALSE,
                HomeEnable     := FALSE
            );
            fbCamSwitchPulserSearch.IN := FALSE;
            fbCamSwitchPulserSync.IN := TRUE;
            nTestStep := 3;
        END_IF

    3: // Restore forward limit after event
        IF fbCamSwitchPulserSync.Q THEN
            fbMotionStage.EnableLimits(
                BackwardEnable := TRUE, 
                ForwardEnable  := TRUE,
                HomeEnable     := FALSE
            );
            fbCamSwitchPulserSync.IN := FALSE;
            nTestStep := 4;
        END_IF

    4: // Wait for "first stage" (positive limit) homing done (i.e. LimHomeDone signals)
        IF fbMotionStage.stExMotionStatus.bLimHomeDone THEN
            // prepare for home switch pulse
            fbCamSwitchPulserSearch.IN := TRUE;
            fbCamSwitchPulserSync.IN := FALSE;
            nTestStep := 5;
        END_IF

    5: // Simulate home switch engagement (simulate HomeEnable = TRUE)
        IF fbCamSwitchPulserSearch.Q THEN
            fbMotionStage.EnableLimits(
                BackwardEnable := TRUE, 
                ForwardEnable  := TRUE,
                HomeEnable     := TRUE
            );
            fbCamSwitchPulserSearch.IN := FALSE;
            fbCamSwitchPulserSync.IN := TRUE;
            nTestStep := 6;
        END_IF

    6: // Simulate home switch disengagement (return HomeEnable to FALSE)
        IF fbCamSwitchPulserSync.Q THEN
            fbMotionStage.EnableLimits(
                BackwardEnable := TRUE, 
                ForwardEnable  := TRUE,
                HomeEnable     := FALSE
            );
            fbCamSwitchPulserSync.IN := FALSE;
            nTestStep := 7;
        END_IF 

    7: // Wait for overall homing to complete (done)
        IF fbMotionStage.stMotionStatus.bDone THEN
            nTestStep := 8;
        END_IF
END_CASE

// Cyclic calls required for timer and cam events and motion stage
fbCamSwitchPulserSearch();
fbCamSwitchPulserSync();
fbTestTimer();
fbMotionStage();

IF nTestStep = 8 THEN
    AssertTrue(
        Condition := fbAxisRef[14].Status.Homed,
        Message := 'Axis not calibrated #1'
    );
    AssertEquals_LREAL(
        Delta := 0.001,
        Expected := fbMotionStage.stMotionCommand.fHomePosition,
        Actual := fbAxisRef[14].NcToPlc.ActPos,
        Message := 'Position is not the expected #2'
    );
    TEST_FINISHED();
ELSIF fbTestTimer.Q THEN
    AssertTrue(
        Condition := FALSE,
        Message := CONCAT('Timed out at step: ', TO_STRING(nTestStep))
    );
    TEST_FINISHED();
END_IF
END_METHOD

METHOD PRIVATE GivenHomeCmdHomeViaHighModeHomeSwPulseMoveOkThenMoveToUserDefinedHomePosition_Test13
VAR_INST
   fbMotionStage : FB_MotionStageNC(	sName := 'Test13',
                                        AxisRef := fbAxisRef[13],
                                        iMotionLogger := fbMotionLogger[13],
                                        iPersistentDataStorage := fbPersistentDataStorage[13]
                                    ):=(SaveAxisParams := FALSE);
									
    fbTestTimer: TON := (IN:=TRUE, PT:=T#10S);
    fbCamSwitchPulserSearch: TON := (IN:=TRUE, PT:=T#500MS);
    fbCamSwitchPulserSync: TON := (PT:=T#1000MS);
    nTestStep : INT;
END_VAR
TEST(__POUNAME());

CASE nTestStep OF
    0: // Enable all interlocks/limits to be ready for homing
		fbMotionStage.EnableLimits(
			BackwardEnable:=TRUE, 
			ForwardEnable:=TRUE,
			HomeEnable:=FALSE
		);
        fbMotionStage.EnableInterlocks();
        nTestStep := 1;

    1: // Issue home command (to low limit)
        fbMotionStage.Home(HomePosition := 20.0, HomeMode := E_EpicsHomeCmd.HOME_VIA_HIGH);
        nTestStep := 2;

    2: // Simulate limit switch drop/restore with cam switch events
        IF fbCamSwitchPulserSearch.Q THEN
			fbMotionStage.EnableLimits(
				BackwardEnable:=TRUE, 
				ForwardEnable:=TRUE,
				HomeEnable:=TRUE
			);
            fbCamSwitchPulserSearch.IN := FALSE;
            fbCamSwitchPulserSync.IN := TRUE;
            nTestStep := 3;
        END_IF

    3: // Restore limit after cam event
        IF fbCamSwitchPulserSync.Q THEN
			fbMotionStage.EnableLimits(
				BackwardEnable:=TRUE, 
				ForwardEnable:=TRUE,
				HomeEnable:=FALSE
			);
            nTestStep := 4;
        END_IF

    4: // Wait for home sequence completion
        IF fbMotionStage.stMotionStatus.bDone THEN
            nTestStep := 5;
        END_IF
END_CASE

fbCamSwitchPulserSearch();
fbCamSwitchPulserSync();
fbTestTimer();
fbMotionStage();

IF nTestStep = 5 THEN
    AssertTrue(
        Condition := fbAxisRef[13].Status.Homed,
        Message := 'Axis not calibrated #1'
    );
    AssertEquals_LREAL(
        Delta := 0.001,
        Expected := fbMotionStage.stMotionCommand.fHomePosition,
        Actual := fbAxisRef[13].NcToPlc.ActPos,
        Message := 'Position is not the expected #2'
    );
    TEST_FINISHED();
ELSIF fbTestTimer.Q THEN
    AssertTrue(
        Condition := FALSE,
        Message := CONCAT('Timed out at step: ', TO_STRING(nTestStep))
    );
    TEST_FINISHED();
END_IF
END_METHOD

METHOD PRIVATE GivenHomeCmdHomeViaLowModeBackwardSwPulseBeforeHomeSwPulseThenMoveToUserDefinePosition_Test15
VAR_INST
   fbMotionStage : FB_MotionStageNC(	sName := 'Test15',
                                        AxisRef := fbAxisRef[15],
                                        iMotionLogger := fbMotionLogger[15],
                                        iPersistentDataStorage := fbPersistentDataStorage[15]
                                    ) :=(SaveAxisParams := FALSE);
									
    fbTestTimer: TON := (IN:=TRUE, PT:=T#10S);
    fbCamSwitchPulserSearch: TON := (IN:=TRUE, PT:=T#500MS);
    fbCamSwitchPulserSync: TON := (PT:=T#1000MS);
    nTestStep : INT;
END_VAR
TEST(__POUNAME());

CASE nTestStep OF
    0: // Enable all interlocks/limits for initial homing (home switch not active yet!)
        fbMotionStage.EnableLimits(
            BackwardEnable := TRUE, 
            ForwardEnable  := TRUE,
            HomeEnable     := FALSE
        );
        fbMotionStage.EnableInterlocks();
        nTestStep := 1;

    1: // Issue homing command (via high limit, should travel to positive end first)
        fbMotionStage.Home(
            HomePosition := 5.0,
            HomeMode := E_EpicsHomeCmd.HOME_VIA_LOW
        );
        nTestStep := 2;

    2: // Simulate forward limit drop
        IF fbCamSwitchPulserSearch.Q THEN
            fbMotionStage.EnableLimits(
                BackwardEnable := FALSE, 
                ForwardEnable  := TRUE,
                HomeEnable     := FALSE
            );
            fbCamSwitchPulserSearch.IN := FALSE;
            fbCamSwitchPulserSync.IN := TRUE;
            nTestStep := 3;
        END_IF

    3: // Restore forward limit after event
        IF fbCamSwitchPulserSync.Q THEN
            fbMotionStage.EnableLimits(
                BackwardEnable := TRUE, 
                ForwardEnable  := TRUE,
                HomeEnable     := FALSE
            );
            fbCamSwitchPulserSync.IN := FALSE;
            nTestStep := 4;
        END_IF

    4: // Wait for "first stage" (positive limit) homing done (i.e. LimHomeDone signals)
        IF fbMotionStage.stExMotionStatus.bLimHomeDone THEN
            // prepare for home switch pulse
            fbCamSwitchPulserSearch.IN := TRUE;
            fbCamSwitchPulserSync.IN := FALSE;
            nTestStep := 5;
        END_IF

    5: // Simulate home switch engagement (simulate HomeEnable = TRUE)
        IF fbCamSwitchPulserSearch.Q THEN
            fbMotionStage.EnableLimits(
                BackwardEnable := TRUE, 
                ForwardEnable  := TRUE,
                HomeEnable     := TRUE
            );
            fbCamSwitchPulserSearch.IN := FALSE;
            fbCamSwitchPulserSync.IN := TRUE;
            nTestStep := 6;
        END_IF

    6: // Simulate home switch disengagement (return HomeEnable to FALSE)
        IF fbCamSwitchPulserSync.Q THEN
            fbMotionStage.EnableLimits(
                BackwardEnable := TRUE, 
                ForwardEnable  := TRUE,
                HomeEnable     := FALSE
            );
            fbCamSwitchPulserSync.IN := FALSE;
            nTestStep := 7;
        END_IF 

    7: // Wait for overall homing to complete (done)
        IF fbMotionStage.stMotionStatus.bDone THEN
            nTestStep := 8;
        END_IF
END_CASE

// Cyclic calls required for timer and cam events and motion stage
fbCamSwitchPulserSearch();
fbCamSwitchPulserSync();
fbTestTimer();
fbMotionStage();

IF nTestStep = 8 THEN
    AssertTrue(
        Condition := fbAxisRef[15].Status.Homed,
        Message := 'Axis not calibrated #1'
    );
    AssertEquals_LREAL(
        Delta := 0.001,
        Expected := fbMotionStage.stMotionCommand.fHomePosition,
        Actual := fbAxisRef[15].NcToPlc.ActPos,
        Message := 'Position is not the expected #2'
    );
    TEST_FINISHED();
ELSIF fbTestTimer.Q THEN
    AssertTrue(
        Condition := FALSE,
        Message := CONCAT('Timed out at step: ', TO_STRING(nTestStep))
    );
    TEST_FINISHED();
END_IF
END_METHOD

METHOD PRIVATE GivenHomeCmdHomeViaLowModeHomeSwPulseMoveOkThenMoveToUserDefinedHomePosition_Test12
VAR_INST
   fbMotionStage : FB_MotionStageNC(	sName := 'Test12',
                                        AxisRef := fbAxisRef[12],
                                        iMotionLogger := fbMotionLogger[12],
                                        iPersistentDataStorage := fbPersistentDataStorage[12]
                                    ) :=(SaveAxisParams := FALSE);
									
    fbTestTimer: TON := (IN:=TRUE, PT:=T#10S);
    fbCamSwitchPulserSearch: TON := (IN:=TRUE, PT:=T#500MS);
    fbCamSwitchPulserSync: TON := (PT:=T#1000MS);
    nTestStep : INT;
END_VAR
TEST(__POUNAME());

CASE nTestStep OF
    0: // Enable all interlocks/limits to be ready for homing
		fbMotionStage.EnableLimits(
			BackwardEnable:=TRUE, 
			ForwardEnable:=TRUE,
			HomeEnable:=FALSE
		);
        fbMotionStage.EnableInterlocks();
        nTestStep := 1;

    1: // Issue home command (to low limit)
        fbMotionStage.Home(HomePosition := 20.0, HomeMode := E_EpicsHomeCmd.HOME_VIA_LOW);
        nTestStep := 2;

    2: // Simulate limit switch drop/restore with cam switch events
        IF fbCamSwitchPulserSearch.Q THEN
			fbMotionStage.EnableLimits(
				BackwardEnable:=TRUE, 
				ForwardEnable:=TRUE,
				HomeEnable:=TRUE
			);
            fbCamSwitchPulserSearch.IN := FALSE;
            fbCamSwitchPulserSync.IN := TRUE;
            nTestStep := 3;
        END_IF

    3: // Restore limit after cam event
        IF fbCamSwitchPulserSync.Q THEN
			fbMotionStage.EnableLimits(
				BackwardEnable:=TRUE, 
				ForwardEnable:=TRUE,
				HomeEnable:=FALSE
			);
            nTestStep := 4;
        END_IF

    4: // Wait for home sequence completion
        IF fbMotionStage.stMotionStatus.bDone THEN
            nTestStep := 5;
        END_IF
END_CASE

fbCamSwitchPulserSearch();
fbCamSwitchPulserSync();
fbTestTimer();
fbMotionStage();

IF nTestStep = 5 THEN
    AssertTrue(
        Condition := fbAxisRef[12].Status.Homed,
        Message := 'Axis not calibrated #1'
    );
    AssertEquals_LREAL(
        Delta := 0.001,
        Expected := fbMotionStage.stMotionCommand.fHomePosition,
        Actual := fbAxisRef[12].NcToPlc.ActPos,
        Message := 'Position is not the expected #2'
    );
    TEST_FINISHED();
ELSIF fbTestTimer.Q THEN
    AssertTrue(
        Condition := FALSE,
        Message := CONCAT('Timed out at step: ', TO_STRING(nTestStep))
    );
    TEST_FINISHED();
END_IF
END_METHOD

METHOD PRIVATE GivenHomeCmdLowLimitModeAndResetThenAbortHoming_Test16
VAR_INST
   fbMotionStage : FB_MotionStageNC(	sName := 'Test16',
                                        AxisRef := fbAxisRef[16],
                                        iMotionLogger := fbMotionLogger[16],
                                        iPersistentDataStorage := fbPersistentDataStorage[16]
                                    ):=(SaveAxisParams := FALSE);
									
    fbTestTimer: TON := (IN:=TRUE, PT:=T#3S);
    fbResetTimer: TON := (IN:=TRUE, PT:=T#500MS);
    nTestStep : INT;
END_VAR
TEST(__POUNAME());


CASE nTestStep OF
    0: // Enable all interlocks/limits for initial homing (home switch not active yet!)
        fbMotionStage.EnableLimits(
            BackwardEnable := TRUE, 
            ForwardEnable  := TRUE,
            HomeEnable     := FALSE
        );
        fbMotionStage.EnableInterlocks();
        nTestStep := 1;

    1: // Issue homing command (via high limit, should travel to positive end first)
        fbMotionStage.Home(
            HomePosition := 5.0,
            HomeMode := E_EpicsHomeCmd.LOW_LIMIT
        );
        nTestStep := 2;
    2:
        IF fbResetTimer.Q THEN
            fbMotionStage.Reset();
            fbResetTimer.IN := FALSE;
            nTestStep := 3;
        END_IF
    3:
		// resetting a homing sequence will set mc_home into error state
        IF fbMotionStage.stMotionStatus.bDone THEN
            nTestStep := 4;
        END_IF
END_CASE

fbResetTimer();
fbTestTimer();
fbMotionStage();

IF nTestStep = 4 THEN
    TEST_FINISHED();
ELSIF fbTestTimer.Q THEN
    AssertTrue(
        Condition := FALSE,
        Message := CONCAT('Timed out at step: ', TO_STRING(nTestStep))
    );

    TEST_FINISHED();
END_IF
END_METHOD

METHOD PRIVATE GivenHomeCmdLowLimitModeBackwardSwPulseMoveOkThenMoveToUserDefinedHomePosition_Test10
VAR_INST
   fbMotionStage : FB_MotionStageNC(	sName := 'Test10',
                                        AxisRef := fbAxisRef[10],
                                        iMotionLogger := fbMotionLogger[10],
                                        iPersistentDataStorage := fbPersistentDataStorage[10]
                                    ):=(SaveAxisParams := FALSE);
									
    fbTestTimer: TON := (IN:=TRUE, PT:=T#10S);
    fbCamSwitchPulserSearch: TON := (IN:=TRUE, PT:=T#500MS);
    fbCamSwitchPulserSync: TON := (PT:=T#1000MS);
    nTestStep : INT;
END_VAR
TEST(__POUNAME());

CASE nTestStep OF
    0: // Enable all interlocks/limits to be ready for homing
        fbMotionStage.EnableLimits(
			BackwardEnable:=TRUE, 
			ForwardEnable:=TRUE,
			HomeEnable:=FALSE
		);
        fbMotionStage.EnableInterlocks();
        nTestStep := 1;

    1: // Issue home command (to low limit)
        fbMotionStage.Home(HomePosition := 20.0, HomeMode := E_EpicsHomeCmd.LOW_LIMIT);
        nTestStep := 2;

    2: // Simulate limit switch drop/restore with cam switch events
		// simulate limit release
        IF fbCamSwitchPulserSearch.Q THEN
			fbMotionStage.EnableLimits(
				BackwardEnable:=FALSE, 
				ForwardEnable:=TRUE,
				HomeEnable:=FALSE
			);
            fbCamSwitchPulserSearch.IN := FALSE;
            fbCamSwitchPulserSync.IN := TRUE;
            nTestStep := 3;
        END_IF

    3: // Restore limit after cam event
        IF fbCamSwitchPulserSync.Q THEN
			fbMotionStage.EnableLimits(
				BackwardEnable:=TRUE, 
				ForwardEnable:=TRUE,
				HomeEnable:=FALSE
			);
            nTestStep := 4;
        END_IF

    4: // Wait for home sequence completion
        IF fbMotionStage.stMotionStatus.bDone THEN
            nTestStep := 5;
        END_IF
END_CASE

fbCamSwitchPulserSearch();
fbCamSwitchPulserSync();
fbTestTimer();
fbMotionStage();

IF nTestStep = 5 THEN
    AssertTrue(
        Condition := fbAxisRef[10].Status.Homed,
        Message := 'Axis not calibrated #1'
    );
    AssertEquals_LREAL(
        Delta := 0.001,
        Expected := fbMotionStage.stMotionCommand.fHomePosition,
        Actual := fbAxisRef[10].NcToPlc.ActPos,
        Message := 'Position is not the expected #2'
    );
    TEST_FINISHED();
ELSIF fbTestTimer.Q THEN
    AssertTrue(
        Condition := FALSE,
        Message := CONCAT('Timed out at step: ', TO_STRING(nTestStep))
    );
    TEST_FINISHED();
END_IF
END_METHOD

METHOD PRIVATE GivenHomeCmdNoneAndMoveOkThenSetHomeFlag_Test9
VAR_INST
   fbMotionStage : FB_MotionStageNC(	sName := 'Test9',
                                        AxisRef := fbAxisRef[9],
                                        iMotionLogger := fbMotionLogger[9],
                                        iPersistentDataStorage := fbPersistentDataStorage[9]
                                    ):=(SaveAxisParams := FALSE);
									
    fbTestTimer: TON := (IN:=TRUE, PT:=T#3S);
    nTestStep : INT;
END_VAR
TEST(__POUNAME());


CASE nTestStep OF
    0:
		// Enable safety interlocks and hardware limits
        fbMotionStage.EnableLimits(
			BackwardEnable:=TRUE, 
			ForwardEnable:=TRUE,
			HomeEnable:=FALSE
		);
        fbMotionStage.EnableInterlocks();
		nTestStep := 1;
	1:
		fbMotionStage.Home(HomePosition:=20.0, HomeMode:=E_EPicsHomeCmd.NONE);
		nTestStep := 2;
	2:
		IF fbMotionStage.stMotionStatus.bHomed THEN
			nTestStep := 3;
		END_IF	
END_CASE

fbTestTimer();
fbMotionStage();

IF nTestStep = 3 THEN

TEST_FINISHED();
ELSIF fbTestTimer.Q THEN
    AssertTrue(
        Condition := FALSE,
        Message := CONCAT('Timed out at step: ', TO_STRING(nTestStep))
    );
    TEST_FINISHED();
END_IF
END_METHOD

METHOD PRIVATE GivenMoveCmdAndMoveOkAndNegativeBacklashEnabledThenMoveToTargetWithCompensation_Test7
VAR_INST
   fbMotionStage : FB_MotionStageNC(	sName := 'Test7',
                                        AxisRef := fbAxisRef[7],
                                        iMotionLogger := fbMotionLogger[7],
                                        iPersistentDataStorage := fbPersistentDataStorage[7]
                                    ):=(SaveAxisParams := FALSE);
									
    fbTestTimer: TON := (IN:=TRUE, PT:=T#10S);
    nTestStep : INT;
END_VAR
TEST(__POUNAME());

CASE nTestStep OF
    0: // Enable safety and backlash compensation
         fbMotionStage.EnableLimits(
			BackwardEnable:=TRUE, 
			ForwardEnable:=TRUE,
			HomeEnable:=FALSE
		);
        fbMotionStage.EnableInterlocks();
		fbMotionStage.EnableBacklashCompensation(UserEnable := TRUE, Compensation := -2.5);
        nTestStep := 1;
    1: // Forward move, should have **no** compensation applied
        fbMotionStage.AbsoluteMoveWithBacklashCompensation(
            Position := -10.0,
            Velocity := 200.0,
            Acceleration := 400.0,
            Deceleration := 400.0
        );
        nTestStep := 2;
    2:
        IF fbMotionStage.stMotionStatus.bDone THEN
            AssertTrue(
                Condition := ABS(-10.0 - fbAxisRef[7].NcToPlc.ActPos) < 0.001,
                Message := 'Target position not reached #1'
            );
            AssertTrue(
                Condition := (fbAxisRef[7].NcToPlc.ActPos - fbAxisRef[7].NcToPlc.ActPosWithoutPosCorrection) = 0,
                Message := 'No compensation in this direction #2'
            );
            nTestStep := 3;
        END_IF
    3: // Reverse move, should have 2.5 compensation
        fbMotionStage.AbsoluteMoveWithBacklashCompensation(
            Position := 80.0,
            Velocity := 200.0,
            Acceleration := 400.0,
            Deceleration := 400.0
        );
        nTestStep := 4;
    4:
        IF fbMotionStage.stMotionStatus.bDone THEN
            AssertTrue(
                Condition := ABS(80.0 - fbAxisRef[7].NcToPlc.ActPos) < 0.001,
                Message := 'Target position not reached #3'
            );
            AssertTrue(
                Condition := (fbAxisRef[7].NcToPlc.ActPos - fbAxisRef[7].NcToPlc.ActPosWithoutPosCorrection) = 2.5,
                Message := 'This move must have a 2.5 compensation #4'
            );
            nTestStep := 5;
        END_IF
    5: // Compensation now 0, move uncompensated
        fbMotionStage.EnableBacklashCompensation(UserEnable := TRUE, Compensation := 0);
        nTestStep := 6;
    6:
        fbMotionStage.AbsoluteMoveWithBacklashCompensation(
            Position := 120.0,
            Velocity := 200.0,
            Acceleration := 400.0,
            Deceleration := 400.0
        );
        nTestStep := 7;
    7:
        IF fbMotionStage.stMotionStatus.bDone THEN
            AssertTrue(
                Condition := ABS(120.0 - fbAxisRef[7].NcToPlc.ActPos) < 0.001,
                Message := 'Target position not reached #5'
            );
            AssertTrue(
                Condition := (fbAxisRef[7].NcToPlc.ActPos - fbAxisRef[7].NcToPlc.ActPosWithoutPosCorrection) = 0,
                Message := 'Actual compensation must be 0 #6'
            );
            nTestStep := 8;
        END_IF
    8: // Set -3.5 for next, expect 3.5 compensation in reverse
        fbMotionStage.EnableBacklashCompensation(UserEnable := TRUE, Compensation := -3.5);
        nTestStep := 9;
    9:
        fbMotionStage.AbsoluteMove(
            Position := 160.0,
            Velocity := 200.0,
            Acceleration := 400.0,
            Deceleration := 400.0
        );
        nTestStep := 10;
    10:
        IF fbMotionStage.stMotionStatus.bDone THEN
            AssertTrue(
                Condition := ABS(160.0 - fbAxisRef[7].NcToPlc.ActPos) < 0.001,
                Message := 'Target position not reached #7'
            );
            AssertTrue(
                Condition := (fbAxisRef[7].NcToPlc.ActPos - fbAxisRef[7].NcToPlc.ActPosWithoutPosCorrection) = 3.5,
                Message := 'This move must have a 3.5 compensation #8'
            );
            nTestStep := 11;
        END_IF
    11: // Disable compensation, next should be uncompensated
        fbMotionStage.EnableBacklashCompensation(UserEnable := FALSE, Compensation := -3.5);
        nTestStep := 12;
    12:
        fbMotionStage.AbsoluteMove(
            Position := 180.0,
            Velocity := 200.0,
            Acceleration := 400.0,
            Deceleration := 400.0
        );
        nTestStep := 13;
    13:
        IF fbMotionStage.stMotionStatus.bDone THEN
            AssertTrue(
                Condition := ABS(180.0 - fbAxisRef[7].NcToPlc.ActPos) < 0.001,
                Message := 'Target position not reached #9'
            );
            AssertTrue(
                Condition := (fbAxisRef[7].NcToPlc.ActPos - fbAxisRef[7].NcToPlc.ActPosWithoutPosCorrection) = 0,
                Message := 'This move is not compensated #10'
            );
            nTestStep := 14;
        END_IF
END_CASE

fbTestTimer();
fbMotionStage();

IF nTestStep = 14 THEN
    TEST_FINISHED();
ELSIF fbTestTimer.Q THEN
    AssertTrue(
        Condition := FALSE,
        Message := CONCAT('Timed out at step: ', TO_STRING(nTestStep))
    );
    TEST_FINISHED();
END_IF
END_METHOD

METHOD PRIVATE GivenMoveCmdAndMoveOkAndPositiveBacklashEnabledThenMoveToTargetWithCompensation_Test6
VAR_INST
   fbMotionStage : FB_MotionStageNC(	sName := 'Test6',
                                        AxisRef := fbAxisRef[6],
                                        iMotionLogger := fbMotionLogger[6],
                                        iPersistentDataStorage := fbPersistentDataStorage[6]
                                    ) :=(SaveAxisParams := FALSE);
									
    fbTestTimer: TON := (IN:=TRUE, PT:=T#10S);
    nTestStep : INT;
END_VAR
TEST(__POUNAME());

CASE nTestStep OF
    0: 
		//Enable safety interlocks AND hardware limits
         fbMotionStage.EnableLimits(
			BackwardEnable:=TRUE, 
			ForwardEnable:=TRUE,
			HomeEnable:=FALSE
		);
		// disable restore saved position
        fbMotionStage.EnableInterlocks();
		//Enable 2.5 backlash compensation
        fbMotionStage.EnableBacklashCompensation(UserEnable := TRUE, Compensation := 2.5);
        nTestStep := 1;
    1: // Forward move, should have **no** compensation applied
        fbMotionStage.AbsoluteMoveWithBacklashCompensation(
            Position := 100.0,
            Velocity := 50.0,
            Acceleration := 500.0,
            Deceleration := 500.0
        );
        nTestStep := 2;
    2: // Wait for move done, check result
        IF fbMotionStage.stMotionStatus.bDone THEN
            AssertTrue(
                Condition := ABS(fbMotionStage.MotionCmd.fPosition - fbAxisRef[6].NcToPlc.ActPos) < 0.001,
                Message := 'Target position not reached #1'
            );
            AssertTrue(
                Condition := (fbAxisRef[6].NcToPlc.ActPos - fbAxisRef[6].NcToPlc.ActPosWithoutPosCorrection) = 0,
                Message := 'No compensation in this direction #2'
            );
            nTestStep := 3;
        END_IF
    3: // Reverse move, should have 2.5 compensation applied
        IF fbMotionStage.ExMotionStatus.bIdling THEN
            fbMotionStage.AbsoluteMoveWithBacklashCompensation(
                Position := 50.0,
                Velocity := 50.0,
                Acceleration := 500.0,
                Deceleration := 500.0
            );
            nTestStep := 4;
        END_IF
    4:
        IF fbMotionStage.stMotionStatus.bDone THEN
            AssertTrue(
                Condition := ABS(fbMotionStage.MotionCmd.fPosition - fbAxisRef[6].NcToPlc.ActPos) < 0.001,
                Message := 'Target position not reached #3'
            );
            AssertTrue(
                Condition := ((fbAxisRef[6].NcToPlc.ActPos - fbAxisRef[6].NcToPlc.ActPosWithoutPosCorrection)- 2.5) < 0.001,
                Message := 'This move must have a 2.5 compensation #4'
            );
            nTestStep := 5;
        END_IF
    5: // Set compensation to 0, next move should be uncompensated
        fbMotionStage.EnableBacklashCompensation(UserEnable := TRUE, Compensation := 0);
        nTestStep := 6;
    6:
        fbMotionStage.AbsoluteMoveWithBacklashCompensation(
            Position := 60.0,
            Velocity := 50.0,
            Acceleration := 200.0,
            Deceleration := 200.0
        );
        nTestStep := 7;
    7:
        IF fbMotionStage.stMotionStatus.bDone THEN
            AssertTrue(
                Condition := ABS(60.0 - fbAxisRef[6].NcToPlc.ActPos) < 0.001,
                Message := 'Target position not reached #5'
            );
            AssertTrue(
                Condition := (fbAxisRef[6].NcToPlc.ActPos - fbAxisRef[6].NcToPlc.ActPosWithoutPosCorrection) = 0,
                Message := 'Actual compensation must be 0 #6'
            );
            nTestStep := 8;
        END_IF
    8: // Set comp to 3.5 for next move
        fbMotionStage.EnableBacklashCompensation(UserEnable := TRUE, Compensation := 3.5);
        nTestStep := 9;
    9:
        fbMotionStage.AbsoluteMoveWithBacklashCompensation(
            Position := 40.0,
            Velocity := 50.0,
            Acceleration := 200.0,
            Deceleration := 200.0
        );
        nTestStep := 10;
    10:
        IF fbMotionStage.stMotionStatus.bDone THEN
            AssertTrue(
                Condition := ABS(40.0 - fbAxisRef[6].NcToPlc.ActPos) < 0.001,
                Message := 'Target position not reached #7'
            );
            AssertTrue(
                Condition := ((fbAxisRef[6].NcToPlc.ActPos - fbAxisRef[6].NcToPlc.ActPosWithoutPosCorrection)- 3.5) < 0.001,
                Message := 'This move must have a 3.5 compensation #8'
            );
            nTestStep := 11;
        END_IF
    11: // Disable compensation, next move should show 0 compensation
        fbMotionStage.EnableBacklashCompensation(UserEnable := FALSE, Compensation := 0.5);
        nTestStep := 12;
    12:
        fbMotionStage.AbsoluteMoveWithBacklashCompensation(
            Position := 20.0,
            Velocity := 50.0,
            Acceleration := 200.0,
            Deceleration := 200.0
        );
        nTestStep := 13;
    13:
        IF fbMotionStage.stMotionStatus.bDone THEN
            AssertTrue(
                Condition := ABS(20.0 - fbAxisRef[6].NcToPlc.ActPos) < 0.001,
                Message := 'Target position not reached #9'
            );
            AssertTrue(
                Condition := (fbAxisRef[6].NcToPlc.ActPos - fbAxisRef[6].NcToPlc.ActPosWithoutPosCorrection) = 0,
                Message := 'This move is not compensated #10'
            );
            nTestStep := 14;
        END_IF
END_CASE

fbTestTimer();
fbMotionStage();

IF nTestStep = 14 THEN
    TEST_FINISHED();
ELSIF fbTestTimer.Q THEN
    AssertTrue(
        Condition := FALSE,
        Message := CONCAT('Timed out at step: ', TO_STRING(nTestStep))
    );
    TEST_FINISHED();
END_IF
END_METHOD

METHOD PRIVATE GivenMoveCmdAndMoveOkIfHaltThenAbortMove_Test2
VAR_INST
   fbMotionStage : FB_MotionStageNC(	sName := 'Test2',
                                        AxisRef := fbAxisRef[2],
                                        iMotionLogger := fbMotionLogger[2],
                                        iPersistentDataStorage := fbPersistentDataStorage[2]
                                    ) :=(SaveAxisParams := FALSE);
									
    fbTestTimer: TON := (IN:=TRUE, PT:=T#3S);
    fbAbsoluteMoveHaltTimer: TON := (PT:=T#100MS);
    nTestStep : INT;
END_VAR
TEST(__POUNAME());

fbMotionStage(); // Call stage logic cyclically

// State machine for staged assertions
CASE nTestStep OF
    // Interlock error check
    0:
        IF fbMotionStage.ExMotionStatus.bInterlocksError THEN
            AssertTrue(
                Condition := fbMotionStage.stMotionStatus.bError,
                Message   := 'Interlock error must be raised #2'
            );
            AssertEquals_UDINT(
                Expected := 11,
                Actual   := fbMotionStage.stMotionStatus.nErrorId,
                Message  := 'Interlock error code is 11 #3'
            );		
        END_IF
        nTestStep := 1;

    // Reset, enable limits and interlocks
    1:
        fbMotionStage.Reset();
        fbMotionStage.EnableLimits(
			BackwardEnable:=TRUE, 
			ForwardEnable:=TRUE,
			HomeEnable:=FALSE
		);
        fbMotionStage.EnableInterlocks();
        // Compiler shouldn't allow property set if property is get-only 
        // (review behavior: see your original comments).
        nTestStep := 2;	

    // After abort, error should be cleared
    2:
        IF fbMotionStage.ExMotionStatus.bAbortDone THEN
            AssertFalse(
                Condition := fbMotionStage.stMotionStatus.bError,
                Message   := 'Error must cleared #4'
            );
            AssertEquals_UDINT(
                Expected := 0,
                Actual   := fbMotionStage.stMotionStatus.nErrorId,
                Message  := 'error ID must 0 #5'
            );
            nTestStep := 3;	
        END_IF

    // Command an absolute move
    3:
        fbMotionStage.AbsoluteMove(
            Position := 1000.0,
            Velocity := 50.0,
            Acceleration := 200.0,
            Deceleration := 200.0
        );
        fbAbsoluteMoveHaltTimer.IN := TRUE;
        nTestStep := 4;

    // After short timer, send Halt
    4:
        IF fbAbsoluteMoveHaltTimer.Q THEN
            fbMotionStage.Halt();
            fbAbsoluteMoveHaltTimer.IN := FALSE;
            nTestStep := 5;
        END_IF

    // After move finishes, check abort status and flags
    5:
        IF fbMotionStage.ExMotionStatus.bIdling THEN
            AssertTrue(
                Condition := fbMotionStage.ExMotionStatus.bAborted,
                Message   := 'Move must be aborted #8'
            );
            AssertFalse(
                Condition := fbMotionStage.stMotionStatus.bBusy,
                Message   := 'Move request must be canceled #9'
            );
            AssertFalse(
                Condition := fbMotionStage.stExMotionStatus.bExecute,
                Message   := 'Move request must cleared #10'
            );
            nTestStep := 6;
        END_IF	
END_CASE

// Cyclically call timer FBs
fbTestTimer();
fbAbsoluteMoveHaltTimer();

// End test or handle timeout
IF nTestStep = 6 THEN
    TEST_FINISHED();
ELSIF fbTestTimer.Q THEN
    AssertTrue(
        Condition := FALSE,
        Message := CONCAT('Timed out at step: ', TO_STRING(nTestStep))
    );
    TEST_FINISHED();
END_IF
END_METHOD

METHOD PRIVATE GivenMoveCmdAndMoveOkIfResetThenAbortMove_Test1
VAR_INST
   fbMotionStage : FB_MotionStageNC(	sName := 'TEST1',
                                        AxisRef := fbAxisRef[1],
                                        iMotionLogger := fbMotionLogger[1],
                                        iPersistentDataStorage := fbPersistentDataStorage[1]
                                    ):=(SaveAxisParams := FALSE);
									
    fbTestTimer: TON := (IN:=TRUE, PT:=T#3S);
    fbAbsoluteMoveResetTimer: TON := (PT:=T#500MS);
    nTestStep : INT;
END_VAR
TEST(__POUNAME());

// motion stage block
fbMotionStage();

// Main test state machine
CASE nTestStep OF
    // === Interlock Fault Test ===
    0:
        IF fbMotionStage.ExMotionStatus.bInterlocksError THEN
            AssertTrue(
                Condition := fbMotionStage.stMotionStatus.bError,
                Message := 'Interlock error must be raised #1'
            );
            AssertEquals_UDINT(
                Expected := 11,
                Actual := fbMotionStage.stMotionStatus.nErrorId,
                Message := 'Interlock error code is 11 #2'
            );
        END_IF
        nTestStep := nTestStep + 1;
    
    // === Reset and Enable Features ===
    1:
        fbMotionStage.Reset();
        fbMotionStage.EnableLimits(
			BackwardEnable:=TRUE, 
			ForwardEnable:=TRUE,
			HomeEnable:=FALSE
		);
        fbMotionStage.EnableInterlocks();
        // Note: Trying to write to a property with 'GET' only should fail! See notes below.
        // fbMotionStage.MotionStatus.bExecute := TRUE; // Should be forbidden if it's a read-only property

        nTestStep := nTestStep + 1;    

    // === Abort Done/Status Check ===
    2:
        IF fbMotionStage.ExMotionStatus.bAbortDone THEN
            AssertFalse(
                Condition := fbMotionStage.stMotionStatus.bError,
                Message := 'Error must be cleared #3'
            );
            AssertEquals_UDINT(
                Expected := 0,
                Actual := fbMotionStage.stMotionStatus.nErrorId,
                Message := 'error ID must be 0 #4'
            );
            nTestStep := nTestStep + 1;    
        END_IF

    // === Absolute Move Request ===
    3:
        fbMotionStage.AbsoluteMove(
            Position := 10000.0,
            Velocity := 50.0,
            Acceleration := 500.0,
            Deceleration := 500.0
        );
        fbAbsoluteMoveResetTimer.IN := TRUE;
        nTestStep := nTestStep + 1;

    // === Move Reset after Timer ===
    4:
        IF fbAbsoluteMoveResetTimer.Q THEN
            fbMotionStage.Reset();
            fbAbsoluteMoveResetTimer.IN := FALSE;
            nTestStep := nTestStep + 1;
        END_IF

    // === Move Done/Abort Confirmation ===
    5:
        IF fbMotionStage.stExMotionStatus.bAbortDone THEN
            nTestStep := nTestStep + 1;
        END_IF
	6:
		IF fbMotionStage.stExMotionStatus.bAborted THEN
            AssertFalse(
                Condition := fbMotionStage.stMotionStatus.bBusy,
                Message := 'Move request must be canceled #6'
            );
            AssertFalse(
                Condition := fbMotionStage.stExMotionStatus.bExecute,
                Message := 'Move request must be cleared #7'
            );
            nTestStep := nTestStep + 1;
		END_IF
END_CASE

// Update timers
fbTestTimer();
fbAbsoluteMoveResetTimer();

// Test Completion Handlers
IF nTestStep = 7 THEN
    TEST_FINISHED();
ELSIF fbTestTimer.Q THEN
    AssertTrue(
        Condition := FALSE,
        Message := CONCAT('Timed out at step: ', TO_STRING(nTestStep))
    );
    TEST_FINISHED();
END_IF
END_METHOD

METHOD PRIVATE GivenMoveCmdAndMoveOkMoveToTarget1ThenTarget2_Test3
VAR_INST
   fbMotionStage : FB_MotionStageNC(	sName := 'Test3',
                                        AxisRef := fbAxisRef[3],
                                        iMotionLogger := fbMotionLogger[3],
                                        iPersistentDataStorage := fbPersistentDataStorage[3]
                                    ):=(SaveAxisParams := FALSE);
									
    fbTestTimer: TON := (IN:=TRUE, PT:=T#10S);
    nTestStep : INT;
END_VAR
TEST(__POUNAME());

CASE nTestStep OF
    0: // Enable safety interlocks and hardware limits
        fbMotionStage.EnableLimits(
			BackwardEnable:=TRUE, 
			ForwardEnable:=TRUE,
			HomeEnable:=FALSE
		);
        fbMotionStage.EnableInterlocks();
        nTestStep := 1;

    1: // Issue initial absolute move to position 100.0 with no backlash
        fbMotionStage.AbsoluteMove(
            Position := 100.0,
            Velocity := 50.0,
            Acceleration := 500.0,
            Deceleration := 500.0
        );
        nTestStep := 2;

    2: // Wait for move done
        IF fbMotionStage.stMotionStatus.bDone THEN
            AssertTrue(
                Condition := ABS(fbMotionStage.MotionCmd.fPosition - fbAxisRef[3].NcToPlc.ActPos) < 0.001,
                Message := 'Target position not reached #1'
            );
            nTestStep := 3;
        END_IF

    3: // When idling, perform another absolute move
        IF fbMotionStage.ExMotionStatus.bIdling THEN
            fbMotionStage.AbsoluteMove(
                Position := 320.0,
                Velocity := 50.0,
                Acceleration := 500.0,
                Deceleration := 500.0
            );
            nTestStep := 4;
        END_IF

    4: // Wait for second move done
        IF fbMotionStage.stMotionStatus.bDone THEN
            AssertTrue(
                Condition := ABS(fbMotionStage.MotionCmd.fPosition - fbAxisRef[3].NcToPlc.ActPos) < 0.001,
                Message := 'Target position not reached #2'
            );
            nTestStep := 5;
          END_IF

END_CASE

fbTestTimer();
fbMotionStage();

IF nTestStep = 5 THEN
    TEST_FINISHED();
ELSIF fbTestTimer.Q THEN
    AssertTrue(
        Condition := FALSE,
        Message := CONCAT('Timed out at step: ', TO_STRING(nTestStep))
    );
    TEST_FINISHED();
END_IF
END_METHOD

METHOD PRIVATE GivenMoveCmdAndValidInterlocksThenMoveToTarget_Test4
VAR_INST
   fbMotionStage : FB_MotionStageNC(	sName := 'Test4',
                                        AxisRef := fbAxisRef[4],
                                        iMotionLogger := fbMotionLogger[4],
                                        iPersistentDataStorage := fbPersistentDataStorage[4]
                                    ):=(SaveAxisParams := FALSE);
									
    fbTestTimer: TON := (IN:=TRUE, PT:=T#3S);
    nTestStep : INT;
END_VAR
TEST(__POUNAME());

CASE nTestStep OF
    0: // Enable safety interlocks and hardware limits
        fbMotionStage.EnableLimits(
			BackwardEnable:=TRUE, 
			ForwardEnable:=TRUE,
			HomeEnable:=FALSE
		);
        fbMotionStage.EnableInterlocks();
        nTestStep := 1;

    1: // Issue initial absolute move to position 100.0 with no backlash
        fbMotionStage.AbsoluteMove(
            Position := 100.0,
            Velocity := 50.0,
            Acceleration := 500.0,
            Deceleration := 500.0
        );
        nTestStep := 2;

    2: // Wait for move done
        IF fbMotionStage.stMotionStatus.bDone THEN
            AssertTrue(
                Condition := ABS(fbMotionStage.MotionCmd.fPosition - fbAxisRef[4].NcToPlc.ActPos) < 0.001,
                Message := 'Target position not reached #1'
            );
            nTestStep := 3;
        END_IF
END_CASE

fbTestTimer();
fbMotionStage();

IF nTestStep = 3 THEN
    TEST_FINISHED();
ELSIF fbTestTimer.Q THEN
    AssertTrue(
        Condition := FALSE,
        Message := CONCAT('Timed out at step: ', TO_STRING(nTestStep))
    );
    TEST_FINISHED();
END_IF
END_METHOD

METHOD PRIVATE GivenMoveCmdValidInterlockAndWrongMotionParamsThenGotoErrorStateIfResetThenGotoInitState_Test5
VAR_INST
   fbMotionStage : FB_MotionStageNC(	sName := 'Test5',
                                        AxisRef := fbAxisRef[5],
                                        iMotionLogger := fbMotionLogger[5],
                                        iPersistentDataStorage := fbPersistentDataStorage[5]
                                    ):=(SaveAxisParams := FALSE);
									
    fbTestTimer: TON := (IN:=TRUE, PT:=T#3S);
    fbAbsoluteMoveTimer: TON := (PT:=T#50MS);
    nTestStep : INT;
END_VAR
TEST(__POUNAME());

CASE nTestStep OF
    0:
        fbMotionStage.EnableLimits(
			BackwardEnable:=TRUE, 
			ForwardEnable:=TRUE,
			HomeEnable:=FALSE
		);
        fbMotionStage.EnableInterlocks();
        nTestStep := 1;
	1:// Issue initial absolute move to position 100.0 with no backlash
        fbMotionStage.AbsoluteMove(
            Position := 100.0,
            Velocity := 0.0,
            Acceleration := 500.0,
            Deceleration := 500.0
        );
		nTestStep := 2;
	2:
		IF (fbMotionStage.stExMotionStatus.eDriveState=E_MoveState.ERROR) THEN
			nTestStep := 3;
		END_IF
END_CASE
fbMotionStage();
fbTestTimer();
fbAbsoluteMoveTimer();


IF nTestStep = 3 THEN

TEST_FINISHED();
ELSIF fbTestTimer.Q THEN
    AssertTrue(
        Condition := FALSE,
        Message := CONCAT('Timed out at step: ', TO_STRING(nTestStep))
    );
    TEST_FINISHED();
END_IF
END_METHOD

METHOD PRIVATE OverallStageFeaturesAndOperationalTests_Test17
VAR_INST
   fbMotionStage : FB_MotionStageNC(	sName := 'Test17',
                                        AxisRef := fbAxisRef[17],
                                        iMotionLogger := fbMotionLogger[17],
                                        iPersistentDataStorage := fbPersistentDataStorage[17]
                                    ) := (SaveAxisParams := FALSE);
									
    fbTestTimer: TON := (IN:=TRUE, PT:=T#180S);
    fbResetTimer: TON := (IN:=FALSE, PT:=T#500MS);;
	fbInMotionTimer : TON := (IN:=FALSE, PT:=T#800MS);;
    fbCamSwitchPulserSearch : TON := (IN:=FALSE, PT:=T#1000MS);
    fbCamSwitchPulserSync: TON := (IN:=FALSE, PT:=T#2000MS);
    nTestStep : INT;
END_VAR
TEST(__POUNAME());

CASE nTestStep OF

/// ------------ INITIAL SETUP ---------------
0:
    fbMotionStage.EnableLimits(
        BackwardEnable := TRUE, ForwardEnable := TRUE, HomeEnable := FALSE);
    fbMotionStage.EnableInterlocks();
    nTestStep := 1;

/// ------- 3 FAST ABSOLUTE MOVES ------------
/// (All moves <= 50 units, velocities set for sub-second moves)
1:
    fbMotionStage.AbsoluteMove(Position := 10.0, Velocity := 50.0, Acceleration := 200.0, Deceleration := 200.0);
    nTestStep := 2;
2:
    IF fbMotionStage.stMotionStatus.bDone THEN
        AssertTrue(ABS(10.0 - fbAxisRef[17].NcToPlc.ActPos) < 0.01, 'Move#1');
        nTestStep := 3;
    END_IF
3:
    fbMotionStage.AbsoluteMove(Position := -8.0, Velocity := 50.0, Acceleration := 200.0, Deceleration := 200.0);
    nTestStep := 4;
4:
    IF fbMotionStage.stMotionStatus.bDone THEN
        AssertTrue(ABS(-8.0 - fbAxisRef[17].NcToPlc.ActPos) < 0.01, 'Move#2');
        nTestStep := 5;
    END_IF
5:
    fbMotionStage.AbsoluteMove(Position := 15.0, Velocity := 50.0, Acceleration := 150.0, Deceleration := 150.0);
    nTestStep := 6;
6:
    IF fbMotionStage.stMotionStatus.bDone THEN
        AssertTrue(ABS(15.0 - fbAxisRef[17].NcToPlc.ActPos) < 0.01, 'Move#3');
        nTestStep := 7;
    END_IF

/// -------- HALT and RESET POS/NEG ------------

7:
    fbMotionStage.AbsoluteMove(Position := 18.0, Velocity := 70.0, Acceleration := 200.0, Deceleration := 200.0);
    fbInMotionTimer.PT := T#120MS;
    fbInMotionTimer.IN := TRUE;
    nTestStep := 8;
8:
    IF fbMotionStage.stMotionStatus.bBusy AND fbInMotionTimer.Q THEN
        fbMotionStage.Halt();
        fbInMotionTimer.IN := FALSE;
        nTestStep := 9;
    END_IF
9:
    IF fbMotionStage.stExMotionStatus.bAborted THEN
        AssertFalse(fbMotionStage.stMotionStatus.bBusy, 'Halt busy/fwd');
        nTestStep := 10;
    END_IF

10:
    fbMotionStage.AbsoluteMove(Position := -12.0, Velocity := 70.0, Acceleration := 200.0, Deceleration := 200.0);
    fbInMotionTimer.PT := T#120MS;
    fbInMotionTimer.IN := TRUE;
    nTestStep := 11;
11:
    IF fbMotionStage.stMotionStatus.bBusy AND fbInMotionTimer.Q THEN
        fbMotionStage.Halt();
        fbInMotionTimer.IN := FALSE;
        nTestStep := 12;
    END_IF
12:
    IF fbMotionStage.stExMotionStatus.bAborted THEN
        AssertFalse(fbMotionStage.stMotionStatus.bBusy, 'Halt busy/bwd');
        nTestStep := 13;
    END_IF

13:
    fbMotionStage.AbsoluteMove(Position := 21.0, Velocity := 70.0, Acceleration := 200.0, Deceleration := 200.0);
    fbInMotionTimer.PT := T#120MS;
    fbInMotionTimer.IN := TRUE;
    nTestStep := 14;
14:
    IF fbMotionStage.stMotionStatus.bBusy AND fbInMotionTimer.Q THEN
        fbMotionStage.Reset();
        fbInMotionTimer.IN := FALSE;
        nTestStep := 15;
    END_IF
15:
    IF fbMotionStage.stExMotionStatus.bAborted THEN
        AssertFalse(fbMotionStage.stMotionStatus.bBusy, 'Reset busy/fwd');
        nTestStep := 16;
    END_IF

16:
    fbMotionStage.AbsoluteMove(Position := -22.0, Velocity := 70.0, Acceleration := 200.0, Deceleration := 200.0);
    fbInMotionTimer.PT := T#120MS;
    fbInMotionTimer.IN := TRUE;
    nTestStep := 17;
17:
    IF fbMotionStage.stMotionStatus.bBusy AND fbInMotionTimer.Q THEN
        fbMotionStage.Reset();
        fbInMotionTimer.IN := FALSE;
        nTestStep := 18;
    END_IF
18:
    IF fbMotionStage.stExMotionStatus.bAborted THEN
        AssertFalse(fbMotionStage.stMotionStatus.bBusy, 'Reset busy/bwd');
        nTestStep := 19;
    END_IF

/// -------- LIMIT HIT TEST (FORWARD THEN BACKWARD) ----------
19:
    fbMotionStage.AbsoluteMove(Position := 25.0, Velocity := 50.0, Acceleration := 120.0, Deceleration := 120.0);
    fbInMotionTimer.PT := T#120MS; fbInMotionTimer.IN := TRUE; nTestStep := 20;
20:
    IF fbMotionStage.stMotionStatus.bBusy AND fbInMotionTimer.Q THEN
        fbMotionStage.EnableLimits(BackwardEnable := TRUE, ForwardEnable := FALSE, HomeEnable := FALSE);
        fbInMotionTimer.IN := FALSE; nTestStep := 21;
    END_IF
21:
    IF fbMotionStage.stMotionStatus.bWarning AND fbMotionStage.stExMotionStatus.bAborted THEN
        fbMotionStage.EnableLimits(BackwardEnable := TRUE, ForwardEnable := TRUE, HomeEnable := FALSE);
        nTestStep := 22;
    END_IF
22: nTestStep := 23;

23:
    fbMotionStage.AbsoluteMove(Position := -25.0, Velocity := 50.0, Acceleration := 120.0, Deceleration := 120.0);
    fbInMotionTimer.PT := T#120MS; fbInMotionTimer.IN := TRUE; nTestStep := 24;
24:
    IF fbMotionStage.stMotionStatus.bBusy AND fbInMotionTimer.Q THEN
        fbMotionStage.EnableLimits(BackwardEnable := FALSE, ForwardEnable := TRUE, HomeEnable := FALSE);
        fbInMotionTimer.IN := FALSE; nTestStep := 25;
    END_IF
25:
    IF fbMotionStage.stMotionStatus.bWarning AND fbMotionStage.stExMotionStatus.bAborted THEN
        fbMotionStage.EnableLimits(BackwardEnable := TRUE, ForwardEnable := TRUE, HomeEnable := FALSE);
        nTestStep := 26;
    END_IF
26: nTestStep := 27;

/// ------------- Home+Move Alternation: All major home modes ------------
/// (Home, then absolute move. All positions ~10-30 units, velocities >= 50.)
27:
    fbMotionStage.Home(HomePosition := 10.0, HomeMode := E_EpicsHomeCmd.LOW_LIMIT);
    fbCamSwitchPulserSearch.IN := TRUE; nTestStep := 28;
28:
    IF fbCamSwitchPulserSearch.Q THEN
        fbMotionStage.EnableLimits(BackwardEnable := FALSE, ForwardEnable := TRUE, HomeEnable := FALSE);
        fbCamSwitchPulserSearch.IN := FALSE; fbCamSwitchPulserSync.IN := TRUE;
        nTestStep := 29;
    END_IF
29:
    IF fbCamSwitchPulserSync.Q THEN
        fbMotionStage.EnableLimits(BackwardEnable := TRUE, ForwardEnable := TRUE, HomeEnable := FALSE);
        fbCamSwitchPulserSync.IN := FALSE; nTestStep := 30;
    END_IF
30:
    IF fbMotionStage.stMotionStatus.bDone THEN
        AssertTrue(fbAxisRef[17].Status.Homed, 'Home#1 (LOW_LIMIT): Axis not calibrated'); 
		AssertEquals_LREAL(Delta := 0.001, Expected := 10.0, Actual := fbAxisRef[17].NcToPlc.ActPos, Message :='Home#1: Not at expected home');
        nTestStep := 31;
    END_IF
31: 
	fbMotionStage.AbsoluteMove(Position := 20.0, Velocity := 50.0, Acceleration := 200.0, Deceleration := 200.0);
	nTestStep := 32;
32: 
	IF fbMotionStage.stMotionStatus.bDone THEN
		AssertTrue(ABS(20.0 - fbAxisRef[17].NcToPlc.ActPos) < 0.01, 'Move#4: Target position not reached after home');
		nTestStep := 33;
	END_IF

33: 
	fbMotionStage.Home(HomePosition := 25.0, HomeMode := E_EpicsHomeCmd.HIGH_LIMIT);
	fbCamSwitchPulserSearch.IN := TRUE; 
	nTestStep := 34;
34: 
	IF fbCamSwitchPulserSearch.Q THEN 
		fbMotionStage.EnableLimits(BackwardEnable := TRUE, ForwardEnable := FALSE, HomeEnable := FALSE);
		fbCamSwitchPulserSearch.IN := FALSE;
		fbCamSwitchPulserSync.IN := TRUE;
		nTestStep := 35;
	END_IF
35: 
	IF fbCamSwitchPulserSync.Q THEN
		fbMotionStage.EnableLimits(BackwardEnable := TRUE, ForwardEnable := TRUE, HomeEnable := FALSE);
		fbCamSwitchPulserSync.IN := FALSE;
		nTestStep := 36;
	END_IF
36: 
	IF fbMotionStage.stMotionStatus.bDone THEN 
		AssertTrue(fbAxisRef[17].Status.Homed, 'Home#2 (HIGH_LIMIT): Axis not calibrated');
		AssertEquals_LREAL(Delta := 0.001, Expected := 25.0, Actual := fbAxisRef[17].NcToPlc.ActPos, Message := 'Home#2: Not at expected home'); 
		nTestStep := 37; 
	END_IF
37: 
	fbMotionStage.AbsoluteMove(Position := -20.0, Velocity := 50.0, Acceleration := 200.0, Deceleration := 200.0); 
	nTestStep := 38;
38: 
	IF fbMotionStage.stMotionStatus.bDone THEN 
		AssertTrue(ABS(-20.0 - fbAxisRef[17].NcToPlc.ActPos) < 0.01, 'Move#5: Target position not reached after home');
		nTestStep := 39; 
	END_IF

39:
    fbMotionStage.Home(HomePosition := 12.0, HomeMode := E_EpicsHomeCmd.HOME_VIA_LOW);
    fbCamSwitchPulserSearch.IN := TRUE; nTestStep := 40;
40: 
	IF fbCamSwitchPulserSearch.Q THEN 
		fbMotionStage.EnableLimits(BackwardEnable := FALSE, ForwardEnable := TRUE, HomeEnable := FALSE); 
		fbCamSwitchPulserSearch.IN := FALSE; 
		fbCamSwitchPulserSync.IN := TRUE; 
		nTestStep := 41; 
	END_IF
41: 
	IF fbCamSwitchPulserSync.Q THEN
		fbMotionStage.EnableLimits(BackwardEnable := TRUE, ForwardEnable := TRUE, HomeEnable := FALSE);
		fbCamSwitchPulserSync.IN := FALSE;
		fbCamSwitchPulserSearch.IN := TRUE;
		nTestStep := 42;
	END_IF
42: 
	IF fbCamSwitchPulserSearch.Q THEN
		fbMotionStage.EnableLimits(BackwardEnable := TRUE, ForwardEnable := TRUE, HomeEnable := TRUE);
		fbCamSwitchPulserSearch.IN := FALSE;
		fbCamSwitchPulserSync.IN := TRUE;
		nTestStep := 43;
	END_IF
43: 
	IF fbCamSwitchPulserSync.Q THEN 
		fbMotionStage.EnableLimits(BackwardEnable := TRUE, ForwardEnable := TRUE, HomeEnable := FALSE);
		fbCamSwitchPulserSync.IN := FALSE; 
		nTestStep := 44; 
	END_IF
44: 
	IF fbMotionStage.stMotionStatus.bDone THEN 
		AssertTrue(fbAxisRef[17].Status.Homed, 'Home#3 (HOME_VIA_LOW): Axis not calibrated'); 
		AssertEquals_LREAL(Delta := 0.001, Expected := 12.0, Actual := fbAxisRef[17].NcToPlc.ActPos, Message := 'Home#3: Not at expected home');
		nTestStep := 45; 
	END_IF
45: 
	fbMotionStage.AbsoluteMove(Position := 25.0, Velocity := 50.0, Acceleration := 200.0, Deceleration := 200.0); 
	nTestStep := 46;
46: 
	IF fbMotionStage.stMotionStatus.bDone THEN 
		AssertTrue(ABS(25.0 - fbAxisRef[17].NcToPlc.ActPos) < 0.01, 'Move#6: Target position not reached after home');
		nTestStep := 47; 
	END_IF

47:
    fbMotionStage.Home(HomePosition := -15.0, HomeMode := E_EpicsHomeCmd.HOME_VIA_HIGH);
    fbCamSwitchPulserSearch.IN := TRUE; nTestStep := 48;
48: 
	IF fbCamSwitchPulserSearch.Q THEN 
		fbMotionStage.EnableLimits(BackwardEnable := TRUE, ForwardEnable := FALSE, HomeEnable := FALSE);
		fbCamSwitchPulserSearch.IN := FALSE;
		fbCamSwitchPulserSync.IN := TRUE;
		nTestStep := 49; 
	END_IF
49: 
	IF fbCamSwitchPulserSync.Q THEN 
		fbMotionStage.EnableLimits(BackwardEnable := TRUE, ForwardEnable := TRUE, HomeEnable := FALSE);
		fbCamSwitchPulserSync.IN := FALSE;
		fbCamSwitchPulserSearch.IN := TRUE;
		nTestStep := 50;
	END_IF
50: 
	IF fbCamSwitchPulserSearch.Q THEN
		fbMotionStage.EnableLimits(BackwardEnable := TRUE, ForwardEnable := TRUE, HomeEnable := TRUE);
		fbCamSwitchPulserSearch.IN := FALSE;
		fbCamSwitchPulserSync.IN := TRUE;
		nTestStep := 51;
	END_IF
51: 
	IF fbCamSwitchPulserSync.Q THEN 
		fbMotionStage.EnableLimits(BackwardEnable := TRUE, ForwardEnable := TRUE, HomeEnable := FALSE);
		fbCamSwitchPulserSync.IN := FALSE;
		nTestStep := 52; 
	END_IF
52: 
	IF fbMotionStage.stMotionStatus.bDone THEN 
		AssertTrue(fbAxisRef[17].Status.Homed, 'Home#4 (HOME_VIA_HIGH): Axis not calibrated');
		AssertEquals_LREAL(Delta := 0.001, Expected := -15.0, Actual := fbAxisRef[17].NcToPlc.ActPos, Message := 'Home#4: Not at expected home');
		nTestStep := 53; 
	END_IF
53: 
	fbMotionStage.AbsoluteMove(Position := -30.0, Velocity := 50.0, Acceleration := 200.0, Deceleration := 200.0);
	nTestStep := 54;
54: 
	IF fbMotionStage.stMotionStatus.bDone THEN 
		AssertTrue(ABS(-30.0 - fbAxisRef[17].NcToPlc.ActPos) < 0.01, 'Move#7: Target position not reached after home'); 
		nTestStep := 55;
	END_IF

55:
    fbMotionStage.Home(HomePosition := 30.0, HomeMode := E_EpicsHomeCmd.ABSOLUTE_SET); 
    nTestStep := 56;
56: 
	IF fbMotionStage.stMotionStatus.bDone THEN 
		AssertTrue(fbAxisRef[17].Status.Homed, 'Home#5 (ABSOLUTE_SET): Axis not calibrated'); 
		AssertEquals_LREAL(Delta := 0.001, Expected := 30.0, Actual := fbAxisRef[17].NcToPlc.ActPos,  Message := 'Home#5: Not at expected home');
		nTestStep := 57; 
	END_IF
57: 
	fbMotionStage.AbsoluteMove(Position := 23.0, Velocity := 50.0, Acceleration := 200.0, Deceleration := 200.0);
	nTestStep := 58;
58: 
	IF fbMotionStage.stMotionStatus.bDone THEN 
		AssertTrue(ABS(23.0 - fbAxisRef[17].NcToPlc.ActPos) < 0.01, 'Move#8: Target position not reached after home');
		nTestStep := 59;
	END_IF

// ---- Backlash Compensation: absolute moves ----
59: 
	fbMotionStage.EnableBacklashCompensation(UserEnable := TRUE, Compensation := 1.2);
	nTestStep := 60;
60: 
	fbMotionStage.AbsoluteMove(Position := 27.5, Velocity := 50.0, Acceleration := 100.0, Deceleration := 100.0);
	nTestStep := 61;
61: 
	IF fbMotionStage.stMotionStatus.bDone THEN 
        AssertTrue(ABS(27.5 - fbAxisRef[17].NcToPlc.ActPos) < 0.01, 'Move#9:No comp fwd expected');
        AssertTrue((fbAxisRef[17].NcToPlc.ActPos - fbAxisRef[17].NcToPlc.ActPosWithoutPosCorrection) = 0.0, 'No compensation in this direction');
        nTestStep := 62; 
    END_IF
62: 
	fbMotionStage.AbsoluteMove(Position := 21.0, Velocity := 50.0, Acceleration := 100.0, Deceleration := 100.0);
	nTestStep := 63;
63: 
	IF fbMotionStage.stMotionStatus.bDone THEN 
        AssertTrue(ABS(21.0 - fbAxisRef[17].NcToPlc.ActPos) < 0.01, 'Move#10: Target not reached'); 
        AssertTrue(((fbAxisRef[17].NcToPlc.ActPos - fbAxisRef[17].NcToPlc.ActPosWithoutPosCorrection)-1.2) < 0.001, 
                   'Compensation 1.2 not applied in reverse'); 
        nTestStep := 64; 
    END_IF
64: 
	fbMotionStage.EnableBacklashCompensation(UserEnable := FALSE, Compensation := 0.0);
	nTestStep := 65;
65: 
	fbMotionStage.AbsoluteMove(Position := -20.0, Velocity := 50.0, Acceleration := 100.0, Deceleration := 100.0);
	nTestStep := 66;
66: 
	IF fbMotionStage.stMotionStatus.bDone THEN 
        AssertTrue(ABS(-20.0 - fbAxisRef[17].NcToPlc.ActPos) < 0.01, 'Move#11: Target not reached (no comp)'); 
        AssertTrue((fbAxisRef[17].NcToPlc.ActPos - fbAxisRef[17].NcToPlc.ActPosWithoutPosCorrection) = 0.0, 'Compensation should be disabled'); 
        nTestStep := 67; 
    END_IF
67: 
	fbMotionStage.EnableBacklashCompensation(UserEnable := TRUE, Compensation := -1.7);
	nTestStep := 68;
68: 
	fbMotionStage.AbsoluteMove(Position := -30.0, Velocity := 50.0, Acceleration := 100.0, Deceleration := 100.0);
	nTestStep := 69;
69: 
	IF fbMotionStage.stMotionStatus.bDone THEN 
        AssertTrue(ABS(-30.0 - fbAxisRef[17].NcToPlc.ActPos) < 0.01, 'Move#12: Target not reached, comp negative'); 
        AssertTrue((fbAxisRef[17].NcToPlc.ActPos - fbAxisRef[17].NcToPlc.ActPosWithoutPosCorrection) = 0.0, 'No comp fwd for neg setting'); 
        nTestStep := 70; 
    END_IF
70: 
	fbMotionStage.AbsoluteMove(Position := 5.0, Velocity := 50.0, Acceleration := 100.0, Deceleration := 100.0);
	nTestStep := 71;
71: 
	IF fbMotionStage.stMotionStatus.bDone THEN 
        AssertTrue(ABS(5.0 - fbAxisRef[17].NcToPlc.ActPos) < 0.01, 'Move#13: Target not reached (comp negative, rev)'); 
        AssertTrue(((fbAxisRef[17].NcToPlc.ActPos - fbAxisRef[17].NcToPlc.ActPosWithoutPosCorrection)-1.7) < 0.001, 'Compensation -1.7 not applied'); 
        nTestStep := 72; 
    END_IF
72:
	fbMotionStage.EnableBacklashCompensation(UserEnable := FALSE, Compensation := 0.0);
	nTestStep := 73;
// --- Absolute Move with ZERO Velocity triggers error ---
73:
    fbMotionStage.AbsoluteMove(
        Position := 10.0,
        Velocity := 0.0,
        Acceleration := 100.0,
        Deceleration := 100.0
    );
    nTestStep := 74;

74:
    IF fbMotionStage.stMotionStatus.bError THEN
        AssertTrue(
            fbMotionStage.stMotionStatus.nErrorId = 16#4359,
            'Not the expected NC error message for zero velocity'
        );
        fbMotionStage.Reset();
        nTestStep := 75;
    END_IF

75:
    IF NOT fbMotionStage.stMotionStatus.bError THEN
        AssertFalse(
            fbMotionStage.stMotionStatus.bError,
            'Error flag should be cleared after reset'
        );
        AssertTrue(
            fbMotionStage.stMotionStatus.sErrorMessage = '',
            'Error message should be cleared after reset'
        );
        nTestStep := 76;
    END_IF

76:
    fbMotionStage.AbsoluteMove(
        Position := 15.0,
        Velocity := 50.0,
        Acceleration := 100.0,
        Deceleration := 100.0
    );
    nTestStep := 77;

77:
    IF fbMotionStage.stMotionStatus.bDone THEN
        AssertTrue(
            ABS(15.0 - fbAxisRef[17].NcToPlc.ActPos) < 0.01,
            'Recovery Move: Target position not reached after valid velocity'
        );
        nTestStep := 78;
    END_IF
END_CASE

